LIN {X -0.033,Y -190.233,Z 1843.877,A 0.000,B 0.000,C 90.000,E1 337.922} C_DIS
LIN {X -0.106,Y -193.186,Z 1843.850,A 0.000,B 0.000,C 90.000,E1 332.999} C_DIS
LIN {X 0.019,Y -196.283,Z 1843.827,A 0.000,B 0.000,C 90.000,E1 328.869} C_DIS
LIN {X -0.019,Y -199.902,Z 1843.804,A 0.000,B 0.000,C 90.000,E1 324.815} C_DIS
LIN {X -0.088,Y -204.049,Z 1843.782,A 0.000,B 0.000,C 90.000,E1 320.803} C_DIS
LIN {X 0.012,Y -209.249,Z 1843.760,A 0.000,B 0.000,C 90.000,E1 316.782} C_DIS
LIN {X -0.006,Y -211.916,Z 1843.751,A 0.000,B 0.000,C 90.000,E1 315.202} C_DIS
LIN {X 0.008,Y -215.116,Z 1843.742,A 0.000,B 0.000,C 90.000,E1 313.623} C_DIS
LIN {X -0.083,Y -218.974,Z 1843.734,A 0.000,B 0.000,C 90.000,E1 312.081} C_DIS
LIN {X -0.117,Y -223.654,Z 1843.725,A 0.000,B 0.000,C 90.000,E1 310.539} C_DIS
LIN {X -0.067,Y -229.271,Z 1843.717,A 0.000,B 0.000,C 90.000,E1 308.991} C_DIS
LIN {X 0.059,Y -235.659,Z 1843.708,A 0.000,B 0.000,C 90.000,E1 307.443} C_DIS
LIN {X -0.053,Y -246.348,Z 1843.696,A 0.000,B 0.000,C 90.000,E1 305.231} C_DIS
LIN {X -0.015,Y -260.231,Z 1843.682,A 0.000,B 0.000,C 90.000,E1 302.673} C_DIS
LIN {X -0.147,Y -278.257,Z 1843.666,A 0.000,B 0.000,C 90.000,E1 299.873} C_DIS
LIN {X -0.079,Y -294.898,Z 1843.652,A 0.000,B 0.000,C 90.000,E1 297.462} C_DIS
LIN {X -0.078,Y -306.901,Z 1843.643,A 0.000,B 0.000,C 90.000,E1 295.796} C_DIS
LIN {X -0.041,Y -323.612,Z 1843.631,A 0.000,B 0.000,C 90.000,E1 293.515} C_DIS
LIN {X 0.188,Y -333.099,Z 1843.624,A 0.000,B 0.000,C 90.000,E1 292.206} C_DIS
LIN {X 0.104,Y -342.269,Z 1843.617,A 0.000,B 0.000,C 90.000,E1 290.972} C_DIS
LIN {X 0.010,Y -350.803,Z 1843.610,A 0.000,B 0.000,C 90.000,E1 289.758} C_DIS
LIN {X -0.017,Y -356.794,Z 1843.605,A 0.000,B 0.000,C 90.000,E1 288.852} C_DIS
LIN {X 0.008,Y -362.167,Z 1843.600,A 0.000,B 0.000,C 90.000,E1 287.946} C_DIS
LIN {X 0.020,Y -365.351,Z 1843.596,A 0.000,B 0.000,C 90.000,E1 287.347} C_DIS
LIN {X 0.131,Y -369.387,Z 1843.591,A 0.000,B 0.000,C 90.000,E1 286.441} C_DIS
LIN {X 0.190,Y -371.679,Z 1843.588,A 0.000,B 0.000,C 90.000,E1 285.843} C_DIS
LIN {X -0.108,Y -374.517,Z 1843.583,A 0.000,B 0.000,C 90.000,E1 285.009} C_DIS
LIN {X -0.025,Y -375.965,Z 1843.580,A 0.000,B 0.000,C 90.000,E1 284.411} C_DIS
LIN {X -0.024,Y -376.991,Z 1843.577,A 0.000,B 0.000,C 90.000,E1 283.828} C_DIS
LIN {X -0.010,Y -377.620,Z 1843.574,A 0.000,B 0.000,C 90.000,E1 283.244} C_DIS
LIN {X 0.094,Y -377.791,Z 1843.570,A 0.000,B 0.000,C 90.000,E1 282.647} C_DIS
LIN {X 0.119,Y -377.552,Z 1843.567,A 0.000,B 0.000,C 90.000,E1 282.063} C_DIS
LIN {X 0.145,Y -376.875,Z 1843.564,A 0.000,B 0.000,C 90.000,E1 281.478} C_DIS
LIN {X 0.170,Y -375.718,Z 1843.561,A 0.000,B 0.000,C 90.000,E1 280.894} C_DIS
LIN {X 0.190,Y -374.108,Z 1843.557,A 0.000,B 0.000,C 90.000,E1 280.310} C_DIS
LIN {X 0.139,Y -370.889,Z 1843.553,A 0.000,B 0.000,C 90.000,E1 279.443} C_DIS
LIN {X -0.018,Y -362.561,Z 1843.541,A 0.000,B 0.000,C 90.000,E1 277.409} C_DIS
LIN {X 0.184,Y -358.290,Z 1843.536,A 0.000,B 0.000,C 90.000,E1 276.486} C_DIS
LIN {X 0.048,Y -354.814,Z 1843.533,A 0.000,B 0.000,C 90.000,E1 275.910} C_DIS
LIN {X -0.105,Y -350.748,Z 1843.530,A 0.000,B 0.000,C 90.000,E1 275.334} C_DIS
LIN {X 0.069,Y -345.924,Z 1843.526,A 0.000,B 0.000,C 90.000,E1 274.702} C_DIS
LIN {X -0.112,Y -340.429,Z 1843.523,A 0.000,B 0.000,C 90.000,E1 274.131} C_DIS
LIN {X -0.087,Y -334.526,Z 1843.520,A 0.000,B 0.000,C 90.000,E1 273.555} C_DIS
LIN {X -0.114,Y -328.400,Z 1843.517,A 0.000,B 0.000,C 90.000,E1 273.037} C_DIS
LIN {X 0.077,Y -322.038,Z 1843.514,A 0.000,B 0.000,C 90.000,E1 272.522} C_DIS
LIN {X -0.131,Y -315.451,Z 1843.512,A 0.000,B 0.000,C 90.000,E1 272.121} C_DIS
LIN {X -0.025,Y -308.681,Z 1843.510,A 0.000,B 0.000,C 90.000,E1 271.718} C_DIS
LIN {X 0.079,Y -301.563,Z 1843.508,A 0.000,B 0.000,C 90.000,E1 271.375} C_DIS
LIN {X -0.137,Y -294.097,Z 1843.506,A 0.000,B 0.000,C 90.000,E1 271.146} C_DIS
LIN {X -0.063,Y -286.185,Z 1843.505,A 0.000,B 0.000,C 90.000,E1 270.917} C_DIS
LIN {X 0.097,Y -271.303,Z 1843.503,A 0.000,B 0.000,C 90.000,E1 270.573} C_DIS
LIN {X 0.056,Y -249.540,Z 1843.501,A 0.000,B 0.000,C 90.000,E1 270.172} C_DIS
LIN {X -0.017,Y -240.784,Z 1843.500,A 0.000,B 0.000,C 90.000,E1 270.057} C_DIS
LIN {X 0.111,Y -230.998,Z 1843.500,A 0.000,B 0.000,C 90.000,E1 269.943} C_DIS
LIN {X 0.068,Y -181.555,Z 1843.500,A 0.000,B 0.000,C 90.000,E1 269.943} C_DIS
LIN {X -0.012,Y -180.816,Z 1843.471,A 0.000,B 0.000,C 90.000,E1 264.837} C_DIS
LIN {X 0.065,Y -178.919,Z 1843.443,A 0.000,B 0.000,C 90.000,E1 259.746} C_DIS
LIN {X -0.026,Y -175.964,Z 1843.415,A 0.000,B 0.000,C 90.000,E1 254.685} C_DIS
LIN {X 0.090,Y -175.441,Z 1843.410,A 0.000,B 0.000,C 90.000,E1 253.795} C_DIS
LIN {X -0.069,Y -172.198,Z 1843.386,A 0.000,B 0.000,C 90.000,E1 249.571} C_DIS
LIN {X -0.092,Y -171.671,Z 1843.382,A 0.000,B 0.000,C 90.000,E1 248.720} C_DIS
LIN {X -0.100,Y -167.896,Z 1843.358,A 0.000,B 0.000,C 90.000,E1 244.409} C_DIS
LIN {X 0.068,Y -166.636,Z 1843.348,A 0.000,B 0.000,C 90.000,E1 242.615} C_DIS
LIN {X -0.026,Y -162.621,Z 1843.324,A 0.000,B 0.000,C 90.000,E1 238.280} C_DIS
LIN {X 0.033,Y -161.307,Z 1843.314,A 0.000,B 0.000,C 90.000,E1 236.501} C_DIS
LIN {X -0.057,Y -157.304,Z 1843.289,A 0.000,B 0.000,C 90.000,E1 232.110} C_DIS
LIN {X 0.096,Y -155.281,Z 1843.275,A 0.000,B 0.000,C 90.000,E1 229.380} C_DIS
LIN {X 0.024,Y -151.646,Z 1843.250,A 0.000,B 0.000,C 90.000,E1 224.919} C_DIS
LIN {X -0.040,Y -150.514,Z 1843.240,A 0.000,B 0.000,C 90.000,E1 223.137} C_DIS
LIN {X -0.016,Y -147.239,Z 1843.214,A 0.000,B 0.000,C 90.000,E1 218.588} C_DIS
LIN {X -0.050,Y -145.263,Z 1843.194,A 0.000,B 0.000,C 90.000,E1 214.945} C_DIS
LIN {X -0.016,Y -142.373,Z 1843.163,A 0.000,B 0.000,C 90.000,E1 209.411} C_DIS
LIN {X -0.021,Y -141.757,Z 1843.153,A 0.000,B 0.000,C 90.000,E1 207.564} C_DIS
LIN {X 0.030,Y -139.498,Z 1843.117,A 0.000,B 0.000,C 90.000,E1 201.046} C_DIS
LIN {X 0.067,Y -139.004,Z 1843.101,A 0.000,B 0.000,C 90.000,E1 198.236} C_DIS
LIN {X 0.023,Y -138.339,Z 1843.055,A 0.000,B 0.000,C 90.000,E1 189.849} C_DIS
LIN {X 0.046,Y -139.406,Z 1843.008,A 0.000,B 0.000,C 90.000,E1 181.432} C_DIS
LIN {X -0.041,Y -141.314,Z 1842.972,A 0.000,B 0.000,C 90.000,E1 174.951} C_DIS
LIN {X 0.057,Y -142.673,Z 1842.956,A 0.000,B 0.000,C 90.000,E1 172.129} C_DIS
LIN {X 0.038,Y -145.026,Z 1842.931,A 0.000,B 0.000,C 90.000,E1 167.521} C_DIS
LIN {X -0.005,Y -147.652,Z 1842.910,A 0.000,B 0.000,C 90.000,E1 163.866} C_DIS
LIN {X -0.070,Y -150.288,Z 1842.890,A 0.000,B 0.000,C 90.000,E1 160.242} C_DIS
LIN {X -0.057,Y -153.695,Z 1842.870,A 0.000,B 0.000,C 90.000,E1 156.613} C_DIS
LIN {X -0.003,Y -157.109,Z 1842.850,A 0.000,B 0.000,C 90.000,E1 152.999} C_DIS
LIN {X 0.074,Y -161.250,Z 1842.830,A 0.000,B 0.000,C 90.000,E1 149.410} C_DIS
LIN {X 0.020,Y -163.337,Z 1842.820,A 0.000,B 0.000,C 90.000,E1 147.661} C_DIS
LIN {X 0.027,Y -167.791,Z 1842.801,A 0.000,B 0.000,C 90.000,E1 144.149} C_DIS
LIN {X 0.043,Y -171.605,Z 1842.786,A 0.000,B 0.000,C 90.000,E1 141.537} C_DIS
LIN {X 0.091,Y -176.559,Z 1842.767,A 0.000,B 0.000,C 90.000,E1 138.081} C_DIS
LIN {X -0.036,Y -180.857,Z 1842.753,A 0.000,B 0.000,C 90.000,E1 135.567} C_DIS
LIN {X -0.052,Y -186.270,Z 1842.734,A 0.000,B 0.000,C 90.000,E1 132.204} C_DIS
LIN {X 0.007,Y -190.905,Z 1842.720,A 0.000,B 0.000,C 90.000,E1 129.688} C_DIS
LIN {X 0.076,Y -196.671,Z 1842.702,A 0.000,B 0.000,C 90.000,E1 126.377} C_DIS
LIN {X -0.006,Y -199.914,Z 1842.693,A 0.000,B 0.000,C 90.000,E1 124.771} C_DIS
LIN {X 0.024,Y -204.306,Z 1842.680,A 0.000,B 0.000,C 90.000,E1 122.339} C_DIS
LIN {X -0.011,Y -210.652,Z 1842.662,A 0.000,B 0.000,C 90.000,E1 119.155} C_DIS
LIN {X 0.093,Y -216.474,Z 1842.644,A 0.000,B 0.000,C 90.000,E1 115.976} C_DIS
LIN {X -0.090,Y -219.587,Z 1842.636,A 0.000,B 0.000,C 90.000,E1 114.463} C_DIS
LIN {X -0.088,Y -224.053,Z 1842.622,A 0.000,B 0.000,C 90.000,E1 111.897} C_DIS
LIN {X 0.120,Y -283.246,Z 1842.621,A 0.000,B 0.000,C 90.000,E1 111.844} C_DIS
LIN {X 0.108,Y -287.787,Z 1842.621,A 0.000,B 0.000,C 90.000,E1 111.716} C_DIS
LIN {X 0.096,Y -289.851,Z 1842.620,A 0.000,B 0.000,C 90.000,E1 111.589} C_DIS
LIN {X -0.038,Y -292.673,Z 1842.619,A 0.000,B 0.000,C 90.000,E1 111.354} C_DIS
LIN {X 0.109,Y -296.409,Z 1842.616,A 0.000,B 0.000,C 90.000,E1 110.791} C_DIS
LIN {X 0.006,Y -309.662,Z 1842.603,A 0.000,B 0.000,C 90.000,E1 108.489} C_DIS
LIN {X 0.117,Y -324.275,Z 1842.590,A 0.000,B 0.000,C 90.000,E1 106.205} C_DIS
LIN {X -0.145,Y -337.983,Z 1842.580,A 0.000,B 0.000,C 90.000,E1 104.356} C_DIS
LIN {X 0.012,Y -352.877,Z 1842.569,A 0.000,B 0.000,C 90.000,E1 102.479} C_DIS
LIN {X 0.073,Y -371.270,Z 1842.558,A 0.000,B 0.000,C 90.000,E1 100.433} C_DIS
LIN {X 0.155,Y -390.141,Z 1842.548,A 0.000,B 0.000,C 90.000,E1 98.568} C_DIS
LIN {X 0.107,Y -409.354,Z 1842.538,A 0.000,B 0.000,C 90.000,E1 96.891} C_DIS
LIN {X -0.048,Y -431.732,Z 1842.529,A 0.000,B 0.000,C 90.000,E1 95.163} C_DIS
LIN {X 0.106,Y -440.040,Z 1842.525,A 0.000,B 0.000,C 90.000,E1 94.531} C_DIS
LIN {X -0.059,Y -443.726,Z 1842.523,A 0.000,B 0.000,C 90.000,E1 94.131} C_DIS
LIN {X 0.140,Y -445.289,Z 1842.521,A 0.000,B 0.000,C 90.000,E1 93.841} C_DIS
LIN {X -0.135,Y -446.467,Z 1842.520,A 0.000,B 0.000,C 90.000,E1 93.612} C_DIS
LIN {X -0.184,Y -447.912,Z 1842.517,A 0.000,B 0.000,C 90.000,E1 93.094} C_DIS
LIN {X 0.197,Y -448.360,Z 1842.514,A 0.000,B 0.000,C 90.000,E1 92.522} C_DIS
LIN {X 0.143,Y -447.881,Z 1842.511,A 0.000,B 0.000,C 90.000,E1 92.007} C_DIS
LIN {X 0.105,Y -446.408,Z 1842.508,A 0.000,B 0.000,C 90.000,E1 91.489} C_DIS
LIN {X -0.145,Y -445.226,Z 1842.507,A 0.000,B 0.000,C 90.000,E1 91.260} C_DIS
LIN {X 0.067,Y -435.424,Z 1842.498,A 0.000,B 0.000,C 90.000,E1 89.656} C_DIS
LIN {X 0.113,Y -425.490,Z 1842.489,A 0.000,B 0.000,C 90.000,E1 88.051} C_DIS
LIN {X 0.084,Y -413.715,Z 1842.479,A 0.000,B 0.000,C 90.000,E1 86.159} C_DIS
LIN {X -0.136,Y -401.847,Z 1842.468,A 0.000,B 0.000,C 90.000,E1 84.261} C_DIS
LIN {X -0.146,Y -389.902,Z 1842.457,A 0.000,B 0.000,C 90.000,E1 82.299} C_DIS
LIN {X 0.018,Y -377.966,Z 1842.446,A 0.000,B 0.000,C 90.000,E1 80.274} C_DIS
LIN {X -0.003,Y -361.271,Z 1842.430,A 0.000,B 0.000,C 90.000,E1 77.353} C_DIS
LIN {X 0.075,Y -345.625,Z 1842.413,A 0.000,B 0.000,C 90.000,E1 74.338} C_DIS
LIN {X 0.111,Y -333.627,Z 1842.399,A 0.000,B 0.000,C 90.000,E1 71.873} C_DIS
LIN {X -0.034,Y -321.887,Z 1842.385,A 0.000,B 0.000,C 90.000,E1 69.390} C_DIS
LIN {X 0.090,Y -309.231,Z 1842.370,A 0.000,B 0.000,C 90.000,E1 66.485} C_DIS
LIN {X 0.059,Y -299.647,Z 1842.357,A 0.000,B 0.000,C 90.000,E1 64.204} C_DIS
LIN {X -0.060,Y -287.547,Z 1842.340,A 0.000,B 0.000,C 90.000,E1 61.229} C_DIS
LIN {X -0.147,Y -278.152,Z 1842.327,A 0.000,B 0.000,C 90.000,E1 58.869} C_DIS
LIN {X -0.011,Y -268.705,Z 1842.313,A 0.000,B 0.000,C 90.000,E1 56.421} C_DIS
LIN {X -0.059,Y -260.529,Z 1842.302,A 0.000,B 0.000,C 90.000,E1 54.322} C_DIS
LIN {X -0.106,Y -252.310,Z 1842.290,A 0.000,B 0.000,C 90.000,E1 52.190} C_DIS
LIN {X -0.005,Y -242.722,Z 1842.276,A 0.000,B 0.000,C 90.000,E1 49.622} C_DIS
LIN {X 0.011,Y -233.304,Z 1842.261,A 0.000,B 0.000,C 90.000,E1 47.025} C_DIS
LIN {X -0.098,Y -222.999,Z 1842.245,A 0.000,B 0.000,C 90.000,E1 44.028} C_DIS
LIN {X 0.023,Y -213.186,Z 1842.227,A 0.000,B 0.000,C 90.000,E1 40.906} C_DIS
LIN {X 0.101,Y -204.177,Z 1842.210,A 0.000,B 0.000,C 90.000,E1 37.729} C_DIS
LIN {X -0.043,Y -200.670,Z 1842.202,A 0.000,B 0.000,C 90.000,E1 36.423} C_DIS
LIN {X 0.097,Y -200.694,Z 1842.202,A 0.000,B 0.000,C 90.000,E1 36.377} C_DIS
LIN {X -0.009,Y -207.756,Z 1842.196,A 0.000,B 0.000,C 90.000,E1 35.358} C_DIS
LIN {X 0.040,Y -209.524,Z 1842.194,A 0.000,B 0.000,C 90.000,E1 34.945} C_DIS
LIN {X 0.089,Y -210.171,Z 1842.192,A 0.000,B 0.000,C 90.000,E1 34.532} C_DIS
LIN {X -0.072,Y -210.542,Z 1842.188,A 0.000,B 0.000,C 90.000,E1 33.785} C_DIS
LIN {X 0.063,Y -210.374,Z 1842.183,A 0.000,B 0.000,C 90.000,E1 32.959} C_DIS
LIN {X 0.041,Y -209.330,Z 1842.174,A 0.000,B 0.000,C 90.000,E1 31.386} C_DIS
LIN {X 0.077,Y -207.876,Z 1842.166,A 0.000,B 0.000,C 90.000,E1 29.795} C_DIS
LIN {X -0.004,Y -205.334,Z 1842.152,A 0.000,B 0.000,C 90.000,E1 27.436} C_DIS
LIN {X -0.011,Y -200.959,Z 1842.130,A 0.000,B 0.000,C 90.000,E1 23.439} C_DIS
LIN {X 0.017,Y -197.151,Z 1842.108,A 0.000,B 0.000,C 90.000,E1 19.396} C_DIS
LIN {X -0.078,Y -193.232,Z 1842.081,A 0.000,B 0.000,C 90.000,E1 14.537} C_DIS
LIN {X 0.049,Y -189.554,Z 1842.049,A 0.000,B 0.000,C 90.000,E1 8.746} C_DIS
LIN {X -0.048,Y -187.048,Z 1842.016,A 0.000,B 0.000,C 90.000,E1 2.980} C_DIS
LIN {X -0.043,Y -185.845,Z 1841.988,A 0.000,B 0.000,C 90.000,E1 357.879} C_DIS
LIN {X 0.070,Y -185.626,Z 1841.956,A 0.000,B 0.000,C 90.000,E1 352.008} C_DIS
LIN {X 0.075,Y -186.651,Z 1841.923,A 0.000,B 0.000,C 90.000,E1 346.172} C_DIS
LIN {X -0.055,Y -188.055,Z 1841.900,A 0.000,B 0.000,C 90.000,E1 342.054} C_DIS
LIN {X 0.061,Y -190.369,Z 1841.873,A 0.000,B 0.000,C 90.000,E1 337.050} C_DIS
LIN {X 0.079,Y -193.498,Z 1841.845,A 0.000,B 0.000,C 90.000,E1 332.103} C_DIS
LIN {X -0.026,Y -196.711,Z 1841.822,A 0.000,B 0.000,C 90.000,E1 328.043} C_DIS
LIN {X -0.050,Y -200.488,Z 1841.800,A 0.000,B 0.000,C 90.000,E1 323.989} C_DIS
LIN {X -0.009,Y -204.833,Z 1841.777,A 0.000,B 0.000,C 90.000,E1 319.952} C_DIS
LIN {X 0.051,Y -209.167,Z 1841.760,A 0.000,B 0.000,C 90.000,E1 316.743} C_DIS
LIN {X 0.116,Y -213.426,Z 1841.747,A 0.000,B 0.000,C 90.000,E1 314.352} C_DIS
LIN {X -0.100,Y -217.998,Z 1841.736,A 0.000,B 0.000,C 90.000,E1 312.447} C_DIS
LIN {X 0.018,Y -222.547,Z 1841.727,A 0.000,B 0.000,C 90.000,E1 310.862} C_DIS
LIN {X -0.054,Y -226.536,Z 1841.721,A 0.000,B 0.000,C 90.000,E1 309.725} C_DIS
LIN {X 0.036,Y -232.619,Z 1841.712,A 0.000,B 0.000,C 90.000,E1 308.177} C_DIS
LIN {X 0.037,Y -241.159,Z 1841.702,A 0.000,B 0.000,C 90.000,E1 306.297} C_DIS
LIN {X -0.115,Y -252.461,Z 1841.689,A 0.000,B 0.000,C 90.000,E1 304.119} C_DIS
LIN {X -0.022,Y -262.758,Z 1841.679,A 0.000,B 0.000,C 90.000,E1 302.291} C_DIS
LIN {X 0.059,Y -281.021,Z 1841.664,A 0.000,B 0.000,C 90.000,E1 299.461} C_DIS
LIN {X 0.069,Y -297.771,Z 1841.651,A 0.000,B 0.000,C 90.000,E1 297.078} C_DIS
LIN {X 0.115,Y -309.796,Z 1841.641,A 0.000,B 0.000,C 90.000,E1 295.412} C_DIS
LIN {X -0.137,Y -324.198,Z 1841.630,A 0.000,B 0.000,C 90.000,E1 293.515} C_DIS
LIN {X 0.097,Y -333.737,Z 1841.623,A 0.000,B 0.000,C 90.000,E1 292.206} C_DIS
LIN {X 0.018,Y -342.918,Z 1841.617,A 0.000,B 0.000,C 90.000,E1 290.972} C_DIS
LIN {X -0.070,Y -351.484,Z 1841.610,A 0.000,B 0.000,C 90.000,E1 289.758} C_DIS
LIN {X -0.092,Y -357.481,Z 1841.605,A 0.000,B 0.000,C 90.000,E1 288.852} C_DIS
LIN {X -0.061,Y -362.841,Z 1841.600,A 0.000,B 0.000,C 90.000,E1 287.946} C_DIS
LIN {X 0.064,Y -366.038,Z 1841.596,A 0.000,B 0.000,C 90.000,E1 287.330} C_DIS
LIN {X 0.098,Y -368.830,Z 1841.593,A 0.000,B 0.000,C 90.000,E1 286.732} C_DIS
LIN {X 0.134,Y -372.332,Z 1841.588,A 0.000,B 0.000,C 90.000,E1 285.843} C_DIS
LIN {X -0.160,Y -375.103,Z 1841.583,A 0.000,B 0.000,C 90.000,E1 285.009} C_DIS
LIN {X -0.072,Y -376.527,Z 1841.580,A 0.000,B 0.000,C 90.000,E1 284.411} C_DIS
LIN {X -0.068,Y -377.488,Z 1841.577,A 0.000,B 0.000,C 90.000,E1 283.828} C_DIS
LIN {X -0.051,Y -378.135,Z 1841.573,A 0.000,B 0.000,C 90.000,E1 283.244} C_DIS
LIN {X 0.057,Y -378.299,Z 1841.570,A 0.000,B 0.000,C 90.000,E1 282.647} C_DIS
LIN {X 0.085,Y -377.992,Z 1841.567,A 0.000,B 0.000,C 90.000,E1 282.063} C_DIS
LIN {X 0.114,Y -377.277,Z 1841.564,A 0.000,B 0.000,C 90.000,E1 281.478} C_DIS
LIN {X 0.141,Y -376.078,Z 1841.561,A 0.000,B 0.000,C 90.000,E1 280.894} C_DIS
LIN {X 0.164,Y -374.447,Z 1841.557,A 0.000,B 0.000,C 90.000,E1 280.310} C_DIS
LIN {X 0.177,Y -372.370,Z 1841.554,A 0.000,B 0.000,C 90.000,E1 279.726} C_DIS
LIN {X -0.034,Y -362.799,Z 1841.541,A 0.000,B 0.000,C 90.000,E1 277.409} C_DIS
LIN {X 0.171,Y -358.476,Z 1841.536,A 0.000,B 0.000,C 90.000,E1 276.486} C_DIS
LIN {X 0.035,Y -355.006,Z 1841.533,A 0.000,B 0.000,C 90.000,E1 275.910} C_DIS
LIN {X -0.115,Y -350.943,Z 1841.530,A 0.000,B 0.000,C 90.000,E1 275.334} C_DIS
LIN {X 0.059,Y -346.104,Z 1841.526,A 0.000,B 0.000,C 90.000,E1 274.702} C_DIS
LIN {X -0.110,Y -340.587,Z 1841.523,A 0.000,B 0.000,C 90.000,E1 274.131} C_DIS
LIN {X -0.072,Y -334.680,Z 1841.520,A 0.000,B 0.000,C 90.000,E1 273.555} C_DIS
LIN {X -0.044,Y -328.746,Z 1841.517,A 0.000,B 0.000,C 90.000,E1 273.037} C_DIS
LIN {X -0.104,Y -322.559,Z 1841.514,A 0.000,B 0.000,C 90.000,E1 272.579} C_DIS
LIN {X 0.028,Y -316.078,Z 1841.512,A 0.000,B 0.000,C 90.000,E1 272.121} C_DIS
LIN {X 0.142,Y -309.263,Z 1841.510,A 0.000,B 0.000,C 90.000,E1 271.718} C_DIS
LIN {X -0.094,Y -302.144,Z 1841.508,A 0.000,B 0.000,C 90.000,E1 271.432} C_DIS
LIN {X -0.058,Y -294.567,Z 1841.506,A 0.000,B 0.000,C 90.000,E1 271.146} C_DIS
LIN {X 0.003,Y -286.661,Z 1841.505,A 0.000,B 0.000,C 90.000,E1 270.917} C_DIS
LIN {X -0.131,Y -271.712,Z 1841.503,A 0.000,B 0.000,C 90.000,E1 270.630} C_DIS
LIN {X 0.114,Y -250.110,Z 1841.501,A 0.000,B 0.000,C 90.000,E1 270.172} C_DIS
LIN {X 0.028,Y -241.287,Z 1841.500,A 0.000,B 0.000,C 90.000,E1 270.057} C_DIS
LIN {X -0.085,Y -231.549,Z 1841.500,A 0.000,B 0.000,C 90.000,E1 270.000} C_DIS
LIN {X -0.087,Y -181.556,Z 1841.500,A 0.000,B 0.000,C 90.000,E1 270.000} C_DIS
LIN {X 0.013,Y -180.819,Z 1841.471,A 0.000,B 0.000,C 90.000,E1 264.837} C_DIS
LIN {X 0.088,Y -178.922,Z 1841.443,A 0.000,B 0.000,C 90.000,E1 259.746} C_DIS
LIN {X -0.002,Y -175.968,Z 1841.415,A 0.000,B 0.000,C 90.000,E1 254.685} C_DIS
LIN {X -0.054,Y -175.448,Z 1841.410,A 0.000,B 0.000,C 90.000,E1 253.850} C_DIS
LIN {X -0.045,Y -172.202,Z 1841.386,A 0.000,B 0.000,C 90.000,E1 249.571} C_DIS
LIN {X -0.068,Y -171.677,Z 1841.382,A 0.000,B 0.000,C 90.000,E1 248.720} C_DIS
LIN {X -0.077,Y -167.903,Z 1841.358,A 0.000,B 0.000,C 90.000,E1 244.409} C_DIS
LIN {X -0.058,Y -166.642,Z 1841.348,A 0.000,B 0.000,C 90.000,E1 242.666} C_DIS
LIN {X -0.003,Y -162.628,Z 1841.324,A 0.000,B 0.000,C 90.000,E1 238.280} C_DIS
LIN {X 0.056,Y -161.315,Z 1841.314,A 0.000,B 0.000,C 90.000,E1 236.501} C_DIS
LIN {X -0.034,Y -157.311,Z 1841.289,A 0.000,B 0.000,C 90.000,E1 232.110} C_DIS
LIN {X -0.101,Y -155.289,Z 1841.275,A 0.000,B 0.000,C 90.000,E1 229.461} C_DIS
LIN {X 0.046,Y -151.651,Z 1841.250,A 0.000,B 0.000,C 90.000,E1 224.919} C_DIS
LIN {X -0.018,Y -150.519,Z 1841.240,A 0.000,B 0.000,C 90.000,E1 223.137} C_DIS
LIN {X 0.006,Y -147.243,Z 1841.214,A 0.000,B 0.000,C 90.000,E1 218.588} C_DIS
LIN {X -0.029,Y -145.268,Z 1841.194,A 0.000,B 0.000,C 90.000,E1 214.945} C_DIS
LIN {X 0.005,Y -142.377,Z 1841.163,A 0.000,B 0.000,C 90.000,E1 209.411} C_DIS
LIN {X 0.054,Y -141.352,Z 1841.148,A 0.000,B 0.000,C 90.000,E1 206.616} C_DIS
LIN {X 0.038,Y -139.339,Z 1841.112,A 0.000,B 0.000,C 90.000,E1 200.120} C_DIS
LIN {X -0.044,Y -139.007,Z 1841.102,A 0.000,B 0.000,C 90.000,E1 198.290} C_DIS
LIN {X 0.044,Y -138.339,Z 1841.055,A 0.000,B 0.000,C 90.000,E1 189.849} C_DIS
LIN {X 0.066,Y -139.403,Z 1841.008,A 0.000,B 0.000,C 90.000,E1 181.432} C_DIS
LIN {X -0.020,Y -141.310,Z 1840.972,A 0.000,B 0.000,C 90.000,E1 174.951} C_DIS
LIN {X -0.063,Y -142.670,Z 1840.956,A 0.000,B 0.000,C 90.000,E1 172.186} C_DIS
LIN {X 0.059,Y -145.020,Z 1840.931,A 0.000,B 0.000,C 90.000,E1 167.521} C_DIS
LIN {X 0.017,Y -147.647,Z 1840.910,A 0.000,B 0.000,C 90.000,E1 163.866} C_DIS
LIN {X -0.048,Y -150.281,Z 1840.890,A 0.000,B 0.000,C 90.000,E1 160.242} C_DIS
LIN {X -0.036,Y -153.686,Z 1840.870,A 0.000,B 0.000,C 90.000,E1 156.613} C_DIS
LIN {X 0.020,Y -157.101,Z 1840.850,A 0.000,B 0.000,C 90.000,E1 152.999} C_DIS
LIN {X -0.042,Y -161.240,Z 1840.830,A 0.000,B 0.000,C 90.000,E1 149.459} C_DIS
LIN {X 0.044,Y -163.327,Z 1840.820,A 0.000,B 0.000,C 90.000,E1 147.661} C_DIS
LIN {X -0.086,Y -167.780,Z 1840.801,A 0.000,B 0.000,C 90.000,E1 144.196} C_DIS
LIN {X 0.065,Y -171.595,Z 1840.786,A 0.000,B 0.000,C 90.000,E1 141.537} C_DIS
LIN {X -0.003,Y -176.547,Z 1840.767,A 0.000,B 0.000,C 90.000,E1 138.119} C_DIS
LIN {X -0.011,Y -180.846,Z 1840.753,A 0.000,B 0.000,C 90.000,E1 135.567} C_DIS
LIN {X -0.027,Y -186.256,Z 1840.734,A 0.000,B 0.000,C 90.000,E1 132.204} C_DIS
LIN {X -0.089,Y -190.893,Z 1840.721,A 0.000,B 0.000,C 90.000,E1 129.725} C_DIS
LIN {X -0.057,Y -196.657,Z 1840.702,A 0.000,B 0.000,C 90.000,E1 126.423} C_DIS
LIN {X 0.019,Y -199.899,Z 1840.693,A 0.000,B 0.000,C 90.000,E1 124.771} C_DIS
LIN {X 0.050,Y -204.292,Z 1840.680,A 0.000,B 0.000,C 90.000,E1 122.339} C_DIS
LIN {X 0.017,Y -210.640,Z 1840.662,A 0.000,B 0.000,C 90.000,E1 119.155} C_DIS
LIN {X 0.120,Y -216.459,Z 1840.645,A 0.000,B 0.000,C 90.000,E1 115.976} C_DIS
LIN {X -0.063,Y -219.576,Z 1840.636,A 0.000,B 0.000,C 90.000,E1 114.463} C_DIS
LIN {X -0.086,Y -224.052,Z 1840.622,A 0.000,B 0.000,C 90.000,E1 111.897} C_DIS
LIN {X 0.119,Y -283.485,Z 1840.621,A 0.000,B 0.000,C 90.000,E1 111.844} C_DIS
LIN {X 0.043,Y -286.450,Z 1840.621,A 0.000,B 0.000,C 90.000,E1 111.791} C_DIS
LIN {X -0.061,Y -290.264,Z 1840.620,A 0.000,B 0.000,C 90.000,E1 111.589} C_DIS
LIN {X -0.002,Y -292.614,Z 1840.619,A 0.000,B 0.000,C 90.000,E1 111.354} C_DIS
LIN {X 0.089,Y -296.429,Z 1840.616,A 0.000,B 0.000,C 90.000,E1 110.791} C_DIS
LIN {X -0.015,Y -309.684,Z 1840.603,A 0.000,B 0.000,C 90.000,E1 108.489} C_DIS
LIN {X 0.095,Y -324.299,Z 1840.590,A 0.000,B 0.000,C 90.000,E1 106.205} C_DIS
LIN {X 0.160,Y -338.009,Z 1840.580,A 0.000,B 0.000,C 90.000,E1 104.300} C_DIS
LIN {X -0.011,Y -352.906,Z 1840.569,A 0.000,B 0.000,C 90.000,E1 102.479} C_DIS
LIN {X 0.052,Y -371.300,Z 1840.558,A 0.000,B 0.000,C 90.000,E1 100.433} C_DIS
LIN {X 0.135,Y -390.172,Z 1840.548,A 0.000,B 0.000,C 90.000,E1 98.568} C_DIS
LIN {X 0.087,Y -409.385,Z 1840.538,A 0.000,B 0.000,C 90.000,E1 96.891} C_DIS
LIN {X -0.067,Y -431.764,Z 1840.529,A 0.000,B 0.000,C 90.000,E1 95.163} C_DIS
LIN {X 0.089,Y -440.063,Z 1840.525,A 0.000,B 0.000,C 90.000,E1 94.531} C_DIS
LIN {X -0.085,Y -443.740,Z 1840.523,A 0.000,B 0.000,C 90.000,E1 94.131} C_DIS
LIN {X 0.114,Y -445.298,Z 1840.521,A 0.000,B 0.000,C 90.000,E1 93.841} C_DIS
LIN {X -0.161,Y -446.470,Z 1840.520,A 0.000,B 0.000,C 90.000,E1 93.612} C_DIS
LIN {X -0.211,Y -447.907,Z 1840.517,A 0.000,B 0.000,C 90.000,E1 93.094} C_DIS
LIN {X 0.170,Y -448.346,Z 1840.514,A 0.000,B 0.000,C 90.000,E1 92.522} C_DIS
LIN {X 0.117,Y -447.860,Z 1840.511,A 0.000,B 0.000,C 90.000,E1 92.007} C_DIS
LIN {X 0.079,Y -446.378,Z 1840.508,A 0.000,B 0.000,C 90.000,E1 91.489} C_DIS
LIN {X -0.171,Y -445.190,Z 1840.507,A 0.000,B 0.000,C 90.000,E1 91.260} C_DIS
LIN {X 0.040,Y -435.384,Z 1840.498,A 0.000,B 0.000,C 90.000,E1 89.656} C_DIS
LIN {X 0.086,Y -425.450,Z 1840.489,A 0.000,B 0.000,C 90.000,E1 88.051} C_DIS
LIN {X 0.057,Y -413.674,Z 1840.479,A 0.000,B 0.000,C 90.000,E1 86.159} C_DIS
LIN {X -0.163,Y -401.804,Z 1840.468,A 0.000,B 0.000,C 90.000,E1 84.261} C_DIS
LIN {X -0.173,Y -389.860,Z 1840.457,A 0.000,B 0.000,C 90.000,E1 82.299} C_DIS
LIN {X -0.009,Y -377.924,Z 1840.446,A 0.000,B 0.000,C 90.000,E1 80.274} C_DIS
LIN {X -0.030,Y -361.229,Z 1840.430,A 0.000,B 0.000,C 90.000,E1 77.353} C_DIS
LIN {X 0.048,Y -345.584,Z 1840.413,A 0.000,B 0.000,C 90.000,E1 74.338} C_DIS
LIN {X 0.084,Y -333.587,Z 1840.399,A 0.000,B 0.000,C 90.000,E1 71.873} C_DIS
LIN {X -0.061,Y -321.843,Z 1840.385,A 0.000,B 0.000,C 90.000,E1 69.390} C_DIS
LIN {X 0.063,Y -309.189,Z 1840.369,A 0.000,B 0.000,C 90.000,E1 66.485} C_DIS
LIN {X 0.032,Y -299.603,Z 1840.357,A 0.000,B 0.000,C 90.000,E1 64.204} C_DIS
LIN {X 0.165,Y -287.502,Z 1840.340,A 0.000,B 0.000,C 90.000,E1 61.179} C_DIS
LIN {X 0.063,Y -278.109,Z 1840.327,A 0.000,B 0.000,C 90.000,E1 58.820} C_DIS
LIN {X -0.037,Y -268.663,Z 1840.313,A 0.000,B 0.000,C 90.000,E1 56.421} C_DIS
LIN {X -0.086,Y -260.488,Z 1840.302,A 0.000,B 0.000,C 90.000,E1 54.322} C_DIS
LIN {X -0.134,Y -252.268,Z 1840.290,A 0.000,B 0.000,C 90.000,E1 52.190} C_DIS
LIN {X -0.032,Y -242.682,Z 1840.276,A 0.000,B 0.000,C 90.000,E1 49.622} C_DIS
LIN {X -0.015,Y -233.263,Z 1840.261,A 0.000,B 0.000,C 90.000,E1 47.025} C_DIS
LIN {X -0.124,Y -222.959,Z 1840.244,A 0.000,B 0.000,C 90.000,E1 44.028} C_DIS
LIN {X -0.003,Y -213.149,Z 1840.227,A 0.000,B 0.000,C 90.000,E1 40.906} C_DIS
LIN {X 0.041,Y -207.133,Z 1840.216,A 0.000,B 0.000,C 90.000,E1 38.830} C_DIS
LIN {X 0.018,Y -207.134,Z 1840.216,A 0.000,B 0.000,C 90.000,E1 38.830} C_DIS
LIN {X 0.080,Y -213.958,Z 1840.210,A 0.000,B 0.000,C 90.000,E1 37.729} C_DIS
LIN {X -0.022,Y -215.625,Z 1840.208,A 0.000,B 0.000,C 90.000,E1 37.363} C_DIS
LIN {X 0.049,Y -216.231,Z 1840.205,A 0.000,B 0.000,C 90.000,E1 36.950} C_DIS
LIN {X 0.044,Y -216.542,Z 1840.201,A 0.000,B 0.000,C 90.000,E1 36.171} C_DIS
LIN {X 0.044,Y -216.336,Z 1840.197,A 0.000,B 0.000,C 90.000,E1 35.391} C_DIS
LIN {X 0.045,Y -215.875,Z 1840.192,A 0.000,B 0.000,C 90.000,E1 34.612} C_DIS
LIN {X -0.083,Y -214.421,Z 1840.184,A 0.000,B 0.000,C 90.000,E1 33.086} C_DIS
LIN {X -0.009,Y -211.580,Z 1840.171,A 0.000,B 0.000,C 90.000,E1 30.718} C_DIS
LIN {X -0.019,Y -208.525,Z 1840.157,A 0.000,B 0.000,C 90.000,E1 28.359} C_DIS
LIN {X 0.087,Y -204.417,Z 1840.140,A 0.000,B 0.000,C 90.000,E1 25.155} C_DIS
LIN {X -0.002,Y -199.841,Z 1840.118,A 0.000,B 0.000,C 90.000,E1 21.173} C_DIS
LIN {X -0.007,Y -195.216,Z 1840.091,A 0.000,B 0.000,C 90.000,E1 16.315} C_DIS
LIN {X -0.055,Y -191.961,Z 1840.068,A 0.000,B 0.000,C 90.000,E1 12.243} C_DIS
LIN {X -0.035,Y -188.799,Z 1840.041,A 0.000,B 0.000,C 90.000,E1 7.296} C_DIS
LIN {X 0.000,Y -185.857,Z 1840.000,A 0.000,B 0.000,C 90.000,E1 360.000} C_DIS
LIN {X -0.057,Y -185.209,Z 1839.960,A 0.000,B 0.000,C 90.000,E1 352.875} C_DIS
LIN {X -0.100,Y -185.876,Z 1839.932,A 0.000,B 0.000,C 90.000,E1 347.881} C_DIS
LIN {X 0.010,Y -187.386,Z 1839.905,A 0.000,B 0.000,C 90.000,E1 342.851} C_DIS
LIN {X 0.096,Y -189.614,Z 1839.877,A 0.000,B 0.000,C 90.000,E1 337.847} C_DIS
LIN {X 0.012,Y -192.673,Z 1839.850,A 0.000,B 0.000,C 90.000,E1 332.922} C_DIS
LIN {X 0.057,Y -196.472,Z 1839.822,A 0.000,B 0.000,C 90.000,E1 327.995} C_DIS
LIN {X 0.137,Y -200.267,Z 1839.800,A 0.000,B 0.000,C 90.000,E1 323.909} C_DIS
LIN {X 0.046,Y -204.669,Z 1839.777,A 0.000,B 0.000,C 90.000,E1 319.908} C_DIS
LIN {X -0.107,Y -207.861,Z 1839.764,A 0.000,B 0.000,C 90.000,E1 317.553} C_DIS
LIN {X -0.073,Y -211.874,Z 1839.751,A 0.000,B 0.000,C 90.000,E1 315.162} C_DIS
LIN {X 0.092,Y -215.166,Z 1839.742,A 0.000,B 0.000,C 90.000,E1 313.542} C_DIS
LIN {X 0.002,Y -219.151,Z 1839.733,A 0.000,B 0.000,C 90.000,E1 312.000} C_DIS
LIN {X -0.029,Y -223.984,Z 1839.725,A 0.000,B 0.000,C 90.000,E1 310.458} C_DIS
LIN {X 0.088,Y -228.205,Z 1839.718,A 0.000,B 0.000,C 90.000,E1 309.277} C_DIS
LIN {X 0.017,Y -236.158,Z 1839.708,A 0.000,B 0.000,C 90.000,E1 307.397} C_DIS
LIN {X -0.081,Y -246.969,Z 1839.695,A 0.000,B 0.000,C 90.000,E1 305.185} C_DIS
LIN {X -0.023,Y -261.007,Z 1839.681,A 0.000,B 0.000,C 90.000,E1 302.625} C_DIS
LIN {X 0.011,Y -279.137,Z 1839.666,A 0.000,B 0.000,C 90.000,E1 299.795} C_DIS
LIN {X 0.104,Y -295.862,Z 1839.652,A 0.000,B 0.000,C 90.000,E1 297.385} C_DIS
LIN {X 0.011,Y -310.339,Z 1839.641,A 0.000,B 0.000,C 90.000,E1 295.412} C_DIS
LIN {X 0.112,Y -324.721,Z 1839.630,A 0.000,B 0.000,C 90.000,E1 293.462} C_DIS
LIN {X 0.054,Y -334.287,Z 1839.623,A 0.000,B 0.000,C 90.000,E1 292.206} C_DIS
LIN {X -0.018,Y -343.514,Z 1839.616,A 0.000,B 0.000,C 90.000,E1 290.972} C_DIS
LIN {X -0.101,Y -352.126,Z 1839.610,A 0.000,B 0.000,C 90.000,E1 289.758} C_DIS
LIN {X -0.117,Y -358.117,Z 1839.605,A 0.000,B 0.000,C 90.000,E1 288.852} C_DIS
LIN {X -0.080,Y -363.491,Z 1839.600,A 0.000,B 0.000,C 90.000,E1 287.946} C_DIS
LIN {X 0.048,Y -366.680,Z 1839.596,A 0.000,B 0.000,C 90.000,E1 287.330} C_DIS
LIN {X 0.086,Y -369.481,Z 1839.593,A 0.000,B 0.000,C 90.000,E1 286.732} C_DIS
LIN {X 0.128,Y -372.939,Z 1839.588,A 0.000,B 0.000,C 90.000,E1 285.843} C_DIS
LIN {X -0.160,Y -375.680,Z 1839.583,A 0.000,B 0.000,C 90.000,E1 285.009} C_DIS
LIN {X -0.069,Y -377.065,Z 1839.580,A 0.000,B 0.000,C 90.000,E1 284.411} C_DIS
LIN {X -0.061,Y -378.030,Z 1839.577,A 0.000,B 0.000,C 90.000,E1 283.828} C_DIS
LIN {X -0.041,Y -378.647,Z 1839.573,A 0.000,B 0.000,C 90.000,E1 283.244} C_DIS
LIN {X 0.071,Y -378.770,Z 1839.570,A 0.000,B 0.000,C 90.000,E1 282.647} C_DIS
LIN {X 0.101,Y -378.462,Z 1839.567,A 0.000,B 0.000,C 90.000,E1 282.063} C_DIS
LIN {X 0.133,Y -377.701,Z 1839.564,A 0.000,B 0.000,C 90.000,E1 281.478} C_DIS
LIN {X 0.164,Y -376.483,Z 1839.561,A 0.000,B 0.000,C 90.000,E1 280.894} C_DIS
LIN {X 0.189,Y -374.806,Z 1839.557,A 0.000,B 0.000,C 90.000,E1 280.310} C_DIS
LIN {X 0.204,Y -372.713,Z 1839.554,A 0.000,B 0.000,C 90.000,E1 279.726} C_DIS
LIN {X 0.025,Y -364.353,Z 1839.543,A 0.000,B 0.000,C 90.000,E1 277.701} C_DIS
LIN {X -0.109,Y -360.307,Z 1839.538,A 0.000,B 0.000,C 90.000,E1 276.834} C_DIS
LIN {X 0.124,Y -357.051,Z 1839.535,A 0.000,B 0.000,C 90.000,E1 276.201} C_DIS
LIN {X -0.015,Y -353.268,Z 1839.531,A 0.000,B 0.000,C 90.000,E1 275.625} C_DIS
LIN {X -0.171,Y -348.796,Z 1839.528,A 0.000,B 0.000,C 90.000,E1 275.049} C_DIS
LIN {X -0.007,Y -343.634,Z 1839.525,A 0.000,B 0.000,C 90.000,E1 274.416} C_DIS
LIN {X -0.135,Y -337.769,Z 1839.521,A 0.000,B 0.000,C 90.000,E1 273.841} C_DIS
LIN {X -0.071,Y -328.831,Z 1839.517,A 0.000,B 0.000,C 90.000,E1 273.037} C_DIS
LIN {X 0.159,Y -322.525,Z 1839.514,A 0.000,B 0.000,C 90.000,E1 272.522} C_DIS
LIN {X -0.027,Y -315.992,Z 1839.512,A 0.000,B 0.000,C 90.000,E1 272.121} C_DIS
LIN {X 0.089,Y -309.189,Z 1839.510,A 0.000,B 0.000,C 90.000,E1 271.718} C_DIS
LIN {X -0.138,Y -302.062,Z 1839.508,A 0.000,B 0.000,C 90.000,E1 271.432} C_DIS
LIN {X -0.069,Y -294.406,Z 1839.506,A 0.000,B 0.000,C 90.000,E1 271.146} C_DIS
LIN {X 0.013,Y -286.689,Z 1839.505,A 0.000,B 0.000,C 90.000,E1 270.917} C_DIS
LIN {X -0.064,Y -275.367,Z 1839.504,A 0.000,B 0.000,C 90.000,E1 270.688} C_DIS
LIN {X -0.118,Y -250.134,Z 1839.501,A 0.000,B 0.000,C 90.000,E1 270.229} C_DIS
LIN {X 0.049,Y -241.308,Z 1839.500,A 0.000,B 0.000,C 90.000,E1 270.057} C_DIS
LIN {X -0.037,Y -232.641,Z 1839.500,A 0.000,B 0.000,C 90.000,E1 270.000} C_DIS
LIN {X -0.063,Y -229.892,Z 1839.500,A 0.000,B 0.000,C 90.000,E1 270.000} C_DIS
LIN {X -0.070,Y -181.557,Z 1839.500,A 0.000,B 0.000,C 90.000,E1 270.000} C_DIS
LIN {X 0.033,Y -180.821,Z 1839.471,A 0.000,B 0.000,C 90.000,E1 264.837} C_DIS
LIN {X -0.067,Y -178.924,Z 1839.443,A 0.000,B 0.000,C 90.000,E1 259.803} C_DIS
LIN {X -0.028,Y -175.971,Z 1839.415,A 0.000,B 0.000,C 90.000,E1 254.700} C_DIS
LIN {X -0.034,Y -175.454,Z 1839.410,A 0.000,B 0.000,C 90.000,E1 253.850} C_DIS
LIN {X -0.026,Y -172.206,Z 1839.386,A 0.000,B 0.000,C 90.000,E1 249.571} C_DIS
LIN {X -0.047,Y -171.681,Z 1839.382,A 0.000,B 0.000,C 90.000,E1 248.720} C_DIS
LIN {X -0.057,Y -167.908,Z 1839.358,A 0.000,B 0.000,C 90.000,E1 244.409} C_DIS
LIN {X -0.038,Y -166.649,Z 1839.348,A 0.000,B 0.000,C 90.000,E1 242.666} C_DIS
LIN {X 0.016,Y -162.632,Z 1839.324,A 0.000,B 0.000,C 90.000,E1 238.280} C_DIS
LIN {X 0.076,Y -161.320,Z 1839.314,A 0.000,B 0.000,C 90.000,E1 236.501} C_DIS
LIN {X -0.016,Y -157.316,Z 1839.289,A 0.000,B 0.000,C 90.000,E1 232.110} C_DIS
LIN {X -0.083,Y -155.296,Z 1839.275,A 0.000,B 0.000,C 90.000,E1 229.461} C_DIS
LIN {X 0.065,Y -151.656,Z 1839.250,A 0.000,B 0.000,C 90.000,E1 224.919} C_DIS
LIN {X 0.001,Y -150.524,Z 1839.240,A 0.000,B 0.000,C 90.000,E1 223.137} C_DIS
LIN {X 0.024,Y -147.248,Z 1839.214,A 0.000,B 0.000,C 90.000,E1 218.588} C_DIS
LIN {X -0.011,Y -145.273,Z 1839.194,A 0.000,B 0.000,C 90.000,E1 214.945} C_DIS
LIN {X 0.023,Y -142.379,Z 1839.163,A 0.000,B 0.000,C 90.000,E1 209.411} C_DIS
LIN {X 0.073,Y -141.355,Z 1839.148,A 0.000,B 0.000,C 90.000,E1 206.616} C_DIS
LIN {X 0.056,Y -139.341,Z 1839.112,A 0.000,B 0.000,C 90.000,E1 200.120} C_DIS
LIN {X -0.026,Y -139.009,Z 1839.102,A 0.000,B 0.000,C 90.000,E1 198.290} C_DIS
LIN {X 0.061,Y -138.340,Z 1839.055,A 0.000,B 0.000,C 90.000,E1 189.849} C_DIS
LIN {X -0.055,Y -139.402,Z 1839.008,A 0.000,B 0.000,C 90.000,E1 181.489} C_DIS
LIN {X -0.002,Y -141.306,Z 1838.972,A 0.000,B 0.000,C 90.000,E1 174.951} C_DIS
LIN {X -0.044,Y -142.668,Z 1838.957,A 0.000,B 0.000,C 90.000,E1 172.186} C_DIS
LIN {X 0.077,Y -145.016,Z 1838.931,A 0.000,B 0.000,C 90.000,E1 167.521} C_DIS
LIN {X 0.035,Y -147.642,Z 1838.910,A 0.000,B 0.000,C 90.000,E1 163.866} C_DIS
LIN {X -0.030,Y -150.276,Z 1838.890,A 0.000,B 0.000,C 90.000,E1 160.242} C_DIS
LIN {X -0.016,Y -153.679,Z 1838.870,A 0.000,B 0.000,C 90.000,E1 156.613} C_DIS
LIN {X 0.040,Y -157.093,Z 1838.850,A 0.000,B 0.000,C 90.000,E1 152.999} C_DIS
LIN {X -0.023,Y -161.231,Z 1838.830,A 0.000,B 0.000,C 90.000,E1 149.459} C_DIS
LIN {X 0.063,Y -163.319,Z 1838.820,A 0.000,B 0.000,C 90.000,E1 147.661} C_DIS
LIN {X -0.066,Y -167.771,Z 1838.801,A 0.000,B 0.000,C 90.000,E1 144.196} C_DIS
LIN {X 0.086,Y -171.586,Z 1838.786,A 0.000,B 0.000,C 90.000,E1 141.537} C_DIS
LIN {X 0.017,Y -176.536,Z 1838.767,A 0.000,B 0.000,C 90.000,E1 138.119} C_DIS
LIN {X 0.010,Y -180.835,Z 1838.753,A 0.000,B 0.000,C 90.000,E1 135.567} C_DIS
LIN {X -0.006,Y -186.244,Z 1838.734,A 0.000,B 0.000,C 90.000,E1 132.204} C_DIS
LIN {X -0.068,Y -190.881,Z 1838.721,A 0.000,B 0.000,C 90.000,E1 129.725} C_DIS
LIN {X -0.036,Y -196.645,Z 1838.702,A 0.000,B 0.000,C 90.000,E1 126.423} C_DIS
LIN {X 0.042,Y -199.885,Z 1838.693,A 0.000,B 0.000,C 90.000,E1 124.771} C_DIS
LIN {X 0.073,Y -204.280,Z 1838.680,A 0.000,B 0.000,C 90.000,E1 122.339} C_DIS
LIN {X 0.039,Y -210.630,Z 1838.662,A 0.000,B 0.000,C 90.000,E1 119.155} C_DIS
LIN {X -0.051,Y -216.448,Z 1838.645,A 0.000,B 0.000,C 90.000,E1 116.027} C_DIS
LIN {X -0.040,Y -219.566,Z 1838.636,A 0.000,B 0.000,C 90.000,E1 114.463} C_DIS
LIN {X -0.090,Y -224.055,Z 1838.622,A 0.000,B 0.000,C 90.000,E1 111.897} C_DIS
LIN {X 0.114,Y -283.757,Z 1838.621,A 0.000,B 0.000,C 90.000,E1 111.844} C_DIS
LIN {X 0.072,Y -286.325,Z 1838.621,A 0.000,B 0.000,C 90.000,E1 111.791} C_DIS
LIN {X -0.031,Y -290.198,Z 1838.620,A 0.000,B 0.000,C 90.000,E1 111.589} C_DIS
LIN {X 0.028,Y -292.564,Z 1838.619,A 0.000,B 0.000,C 90.000,E1 111.354} C_DIS
LIN {X 0.135,Y -296.378,Z 1838.616,A 0.000,B 0.000,C 90.000,E1 110.791} C_DIS
LIN {X 0.032,Y -309.630,Z 1838.603,A 0.000,B 0.000,C 90.000,E1 108.489} C_DIS
LIN {X -0.169,Y -324.239,Z 1838.590,A 0.000,B 0.000,C 90.000,E1 106.260} C_DIS
LIN {X -0.118,Y -337.944,Z 1838.580,A 0.000,B 0.000,C 90.000,E1 104.356} C_DIS
LIN {X 0.039,Y -352.836,Z 1838.569,A 0.000,B 0.000,C 90.000,E1 102.479} C_DIS
LIN {X 0.099,Y -371.228,Z 1838.558,A 0.000,B 0.000,C 90.000,E1 100.433} C_DIS
LIN {X 0.180,Y -390.098,Z 1838.548,A 0.000,B 0.000,C 90.000,E1 98.568} C_DIS
LIN {X 0.131,Y -409.310,Z 1838.538,A 0.000,B 0.000,C 90.000,E1 96.891} C_DIS
LIN {X -0.026,Y -431.688,Z 1838.529,A 0.000,B 0.000,C 90.000,E1 95.163} C_DIS
LIN {X 0.129,Y -439.999,Z 1838.525,A 0.000,B 0.000,C 90.000,E1 94.531} C_DIS
LIN {X -0.035,Y -443.688,Z 1838.523,A 0.000,B 0.000,C 90.000,E1 94.131} C_DIS
LIN {X 0.165,Y -445.254,Z 1838.521,A 0.000,B 0.000,C 90.000,E1 93.841} C_DIS
LIN {X -0.111,Y -446.434,Z 1838.520,A 0.000,B 0.000,C 90.000,E1 93.612} C_DIS
LIN {X -0.160,Y -447.882,Z 1838.517,A 0.000,B 0.000,C 90.000,E1 93.094} C_DIS
LIN {X 0.222,Y -448.333,Z 1838.514,A 0.000,B 0.000,C 90.000,E1 92.522} C_DIS
LIN {X 0.167,Y -447.856,Z 1838.511,A 0.000,B 0.000,C 90.000,E1 92.007} C_DIS
LIN {X 0.129,Y -446.387,Z 1838.508,A 0.000,B 0.000,C 90.000,E1 91.489} C_DIS
LIN {X -0.120,Y -445.207,Z 1838.507,A 0.000,B 0.000,C 90.000,E1 91.260} C_DIS
LIN {X 0.089,Y -435.404,Z 1838.498,A 0.000,B 0.000,C 90.000,E1 89.656} C_DIS
LIN {X 0.135,Y -425.474,Z 1838.489,A 0.000,B 0.000,C 90.000,E1 88.051} C_DIS
LIN {X 0.105,Y -413.697,Z 1838.479,A 0.000,B 0.000,C 90.000,E1 86.159} C_DIS
LIN {X -0.115,Y -401.827,Z 1838.468,A 0.000,B 0.000,C 90.000,E1 84.261} C_DIS
LIN {X -0.127,Y -389.883,Z 1838.457,A 0.000,B 0.000,C 90.000,E1 82.299} C_DIS
LIN {X 0.036,Y -377.947,Z 1838.446,A 0.000,B 0.000,C 90.000,E1 80.274} C_DIS
LIN {X 0.014,Y -361.247,Z 1838.430,A 0.000,B 0.000,C 90.000,E1 77.353} C_DIS
LIN {X 0.090,Y -345.600,Z 1838.413,A 0.000,B 0.000,C 90.000,E1 74.338} C_DIS
LIN {X 0.125,Y -333.600,Z 1838.399,A 0.000,B 0.000,C 90.000,E1 71.873} C_DIS
LIN {X -0.021,Y -321.856,Z 1838.385,A 0.000,B 0.000,C 90.000,E1 69.390} C_DIS
LIN {X 0.102,Y -309.200,Z 1838.370,A 0.000,B 0.000,C 90.000,E1 66.485} C_DIS
LIN {X 0.070,Y -299.610,Z 1838.357,A 0.000,B 0.000,C 90.000,E1 64.204} C_DIS
LIN {X -0.050,Y -287.508,Z 1838.340,A 0.000,B 0.000,C 90.000,E1 61.229} C_DIS
LIN {X -0.139,Y -278.116,Z 1838.327,A 0.000,B 0.000,C 90.000,E1 58.869} C_DIS
LIN {X -0.004,Y -268.671,Z 1838.313,A 0.000,B 0.000,C 90.000,E1 56.421} C_DIS
LIN {X -0.052,Y -260.498,Z 1838.302,A 0.000,B 0.000,C 90.000,E1 54.322} C_DIS
LIN {X -0.101,Y -252.279,Z 1838.290,A 0.000,B 0.000,C 90.000,E1 52.190} C_DIS
LIN {X -0.001,Y -242.692,Z 1838.276,A 0.000,B 0.000,C 90.000,E1 49.622} C_DIS
LIN {X 0.015,Y -233.272,Z 1838.261,A 0.000,B 0.000,C 90.000,E1 47.025} C_DIS
LIN {X -0.095,Y -222.966,Z 1838.245,A 0.000,B 0.000,C 90.000,E1 44.028} C_DIS
LIN {X 0.006,Y -213.872,Z 1838.229,A 0.000,B 0.000,C 90.000,E1 41.148} C_DIS
LIN {X -0.017,Y -213.868,Z 1838.229,A 0.000,B 0.000,C 90.000,E1 41.148} C_DIS
LIN {X -0.024,Y -219.873,Z 1838.223,A 0.000,B 0.000,C 90.000,E1 40.135} C_DIS
LIN {X 0.061,Y -221.779,Z 1838.221,A 0.000,B 0.000,C 90.000,E1 39.725} C_DIS
LIN {X -0.024,Y -222.481,Z 1838.219,A 0.000,B 0.000,C 90.000,E1 39.358} C_DIS
LIN {X -0.027,Y -222.812,Z 1838.214,A 0.000,B 0.000,C 90.000,E1 38.588} C_DIS
LIN {X 0.008,Y -222.549,Z 1838.210,A 0.000,B 0.000,C 90.000,E1 37.810} C_DIS
LIN {X -0.089,Y -221.231,Z 1838.202,A 0.000,B 0.000,C 90.000,E1 36.297} C_DIS
LIN {X -0.124,Y -218.467,Z 1838.189,A 0.000,B 0.000,C 90.000,E1 33.992} C_DIS
LIN {X 0.033,Y -215.119,Z 1838.176,A 0.000,B 0.000,C 90.000,E1 31.623} C_DIS
LIN {X 0.054,Y -210.453,Z 1838.158,A 0.000,B 0.000,C 90.000,E1 28.487} C_DIS
LIN {X 0.108,Y -204.809,Z 1838.136,A 0.000,B 0.000,C 90.000,E1 24.515} C_DIS
LIN {X -0.052,Y -199.954,Z 1838.114,A 0.000,B 0.000,C 90.000,E1 20.556} C_DIS
LIN {X 0.067,Y -195.057,Z 1838.087,A 0.000,B 0.000,C 90.000,E1 15.662} C_DIS
LIN {X -0.032,Y -190.969,Z 1838.060,A 0.000,B 0.000,C 90.000,E1 10.782} C_DIS
LIN {X -0.007,Y -187.279,Z 1838.028,A 0.000,B 0.000,C 90.000,E1 4.992} C_DIS
LIN {X 0.025,Y -184.924,Z 1837.984,A 0.000,B 0.000,C 90.000,E1 357.020} C_DIS
LIN {X -0.054,Y -184.963,Z 1837.951,A 0.000,B 0.000,C 90.000,E1 351.197} C_DIS
LIN {X -0.001,Y -186.194,Z 1837.919,A 0.000,B 0.000,C 90.000,E1 345.338} C_DIS
LIN {X -0.077,Y -188.047,Z 1837.891,A 0.000,B 0.000,C 90.000,E1 340.369} C_DIS
LIN {X 0.066,Y -190.731,Z 1837.863,A 0.000,B 0.000,C 90.000,E1 335.357} C_DIS
LIN {X 0.011,Y -193.573,Z 1837.840,A 0.000,B 0.000,C 90.000,E1 331.257} C_DIS
LIN {X 0.008,Y -196.944,Z 1837.818,A 0.000,B 0.000,C 90.000,E1 327.168} C_DIS
LIN {X -0.061,Y -200.904,Z 1837.795,A 0.000,B 0.000,C 90.000,E1 323.130} C_DIS
LIN {X -0.012,Y -205.525,Z 1837.773,A 0.000,B 0.000,C 90.000,E1 319.094} C_DIS
LIN {X -0.013,Y -209.019,Z 1837.759,A 0.000,B 0.000,C 90.000,E1 316.701} C_DIS
LIN {X 0.115,Y -211.867,Z 1837.751,A 0.000,B 0.000,C 90.000,E1 315.081} C_DIS
LIN {X -0.022,Y -215.205,Z 1837.742,A 0.000,B 0.000,C 90.000,E1 313.542} C_DIS
LIN {X -0.114,Y -219.287,Z 1837.733,A 0.000,B 0.000,C 90.000,E1 312.000} C_DIS
LIN {X -0.069,Y -222.865,Z 1837.727,A 0.000,B 0.000,C 90.000,E1 310.825} C_DIS
LIN {X 0.033,Y -226.942,Z 1837.720,A 0.000,B 0.000,C 90.000,E1 309.644} C_DIS
LIN {X 0.086,Y -234.730,Z 1837.710,A 0.000,B 0.000,C 90.000,E1 307.729} C_DIS
LIN {X -0.042,Y -245.393,Z 1837.697,A 0.000,B 0.000,C 90.000,E1 305.518} C_DIS
LIN {X 0.097,Y -257.236,Z 1837.685,A 0.000,B 0.000,C 90.000,E1 303.293} C_DIS
LIN {X -0.090,Y -268.007,Z 1837.675,A 0.000,B 0.000,C 90.000,E1 301.544} C_DIS
LIN {X 0.032,Y -284.269,Z 1837.662,A 0.000,B 0.000,C 90.000,E1 299.077} C_DIS
LIN {X -0.013,Y -298.761,Z 1837.650,A 0.000,B 0.000,C 90.000,E1 297.052} C_DIS
LIN {X -0.060,Y -313.305,Z 1837.639,A 0.000,B 0.000,C 90.000,E1 295.079} C_DIS
LIN {X 0.038,Y -327.811,Z 1837.629,A 0.000,B 0.000,C 90.000,E1 293.131} C_DIS
LIN {X -0.141,Y -339.702,Z 1837.620,A 0.000,B 0.000,C 90.000,E1 291.589} C_DIS
LIN {X 0.174,Y -348.626,Z 1837.613,A 0.000,B 0.000,C 90.000,E1 290.301} C_DIS
LIN {X 0.128,Y -354.947,Z 1837.608,A 0.000,B 0.000,C 90.000,E1 289.396} C_DIS
LIN {X 0.137,Y -360.705,Z 1837.603,A 0.000,B 0.000,C 90.000,E1 288.489} C_DIS
LIN {X -0.096,Y -364.212,Z 1837.599,A 0.000,B 0.000,C 90.000,E1 287.928} C_DIS
LIN {X -0.076,Y -367.385,Z 1837.596,A 0.000,B 0.000,C 90.000,E1 287.330} C_DIS
LIN {X -0.035,Y -370.172,Z 1837.593,A 0.000,B 0.000,C 90.000,E1 286.732} C_DIS
LIN {X 0.013,Y -373.602,Z 1837.588,A 0.000,B 0.000,C 90.000,E1 285.843} C_DIS
LIN {X 0.094,Y -376.306,Z 1837.583,A 0.000,B 0.000,C 90.000,E1 284.954} C_DIS
LIN {X 0.190,Y -377.649,Z 1837.580,A 0.000,B 0.000,C 90.000,E1 284.356} C_DIS
LIN {X -0.163,Y -378.568,Z 1837.577,A 0.000,B 0.000,C 90.000,E1 283.828} C_DIS
LIN {X -0.141,Y -379.134,Z 1837.573,A 0.000,B 0.000,C 90.000,E1 283.244} C_DIS
LIN {X -0.025,Y -379.236,Z 1837.570,A 0.000,B 0.000,C 90.000,E1 282.647} C_DIS
LIN {X 0.009,Y -378.902,Z 1837.567,A 0.000,B 0.000,C 90.000,E1 282.063} C_DIS
LIN {X 0.044,Y -378.114,Z 1837.564,A 0.000,B 0.000,C 90.000,E1 281.478} C_DIS
LIN {X 0.077,Y -376.868,Z 1837.561,A 0.000,B 0.000,C 90.000,E1 280.894} C_DIS
LIN {X 0.104,Y -375.147,Z 1837.557,A 0.000,B 0.000,C 90.000,E1 280.310} C_DIS
LIN {X 0.065,Y -371.808,Z 1837.552,A 0.000,B 0.000,C 90.000,E1 279.443} C_DIS
LIN {X -0.048,Y -364.596,Z 1837.543,A 0.000,B 0.000,C 90.000,E1 277.701} C_DIS
LIN {X 0.179,Y -360.503,Z 1837.538,A 0.000,B 0.000,C 90.000,E1 276.777} C_DIS
LIN {X 0.057,Y -357.165,Z 1837.535,A 0.000,B 0.000,C 90.000,E1 276.201} C_DIS
LIN {X -0.080,Y -353.393,Z 1837.531,A 0.000,B 0.000,C 90.000,E1 275.625} C_DIS
LIN {X 0.111,Y -348.893,Z 1837.528,A 0.000,B 0.000,C 90.000,E1 274.992} C_DIS
LIN {X -0.069,Y -343.665,Z 1837.524,A 0.000,B 0.000,C 90.000,E1 274.416} C_DIS
LIN {X 0.151,Y -337.850,Z 1837.521,A 0.000,B 0.000,C 90.000,E1 273.784} C_DIS
LIN {X -0.029,Y -331.811,Z 1837.518,A 0.000,B 0.000,C 90.000,E1 273.269} C_DIS
LIN {X 0.067,Y -325.597,Z 1837.515,A 0.000,B 0.000,C 90.000,E1 272.751} C_DIS
LIN {X 0.073,Y -319.043,Z 1837.513,A 0.000,B 0.000,C 90.000,E1 272.293} C_DIS
LIN {X 0.056,Y -312.397,Z 1837.511,A 0.000,B 0.000,C 90.000,E1 271.892} C_DIS
LIN {X 0.010,Y -305.351,Z 1837.509,A 0.000,B 0.000,C 90.000,E1 271.547} C_DIS
LIN {X 0.010,Y -298.388,Z 1837.507,A 0.000,B 0.000,C 90.000,E1 271.260} C_DIS
LIN {X -0.062,Y -290.518,Z 1837.506,A 0.000,B 0.000,C 90.000,E1 271.031} C_DIS
LIN {X 0.025,Y -279.146,Z 1837.504,A 0.000,B 0.000,C 90.000,E1 270.745} C_DIS
LIN {X -0.089,Y -253.606,Z 1837.501,A 0.000,B 0.000,C 90.000,E1 270.286} C_DIS
LIN {X 0.036,Y -240.960,Z 1837.500,A 0.000,B 0.000,C 90.000,E1 270.057} C_DIS
LIN {X 0.007,Y -233.460,Z 1837.500,A 0.000,B 0.000,C 90.000,E1 270.000} C_DIS
LIN {X -0.039,Y -228.868,Z 1837.500,A 0.000,B 0.000,C 90.000,E1 270.000} C_DIS
LIN {X -0.049,Y -181.558,Z 1837.500,A 0.000,B 0.000,C 90.000,E1 270.000} C_DIS
LIN {X 0.060,Y -180.823,Z 1837.471,A 0.000,B 0.000,C 90.000,E1 264.837} C_DIS
LIN {X -0.039,Y -178.927,Z 1837.443,A 0.000,B 0.000,C 90.000,E1 259.803} C_DIS
LIN {X -0.001,Y -175.975,Z 1837.415,A 0.000,B 0.000,C 90.000,E1 254.700} C_DIS
LIN {X -0.056,Y -175.461,Z 1837.410,A 0.000,B 0.000,C 90.000,E1 253.866} C_DIS
LIN {X 0.001,Y -172.212,Z 1837.386,A 0.000,B 0.000,C 90.000,E1 249.571} C_DIS
LIN {X -0.021,Y -171.688,Z 1837.382,A 0.000,B 0.000,C 90.000,E1 248.720} C_DIS
LIN {X -0.030,Y -167.915,Z 1837.358,A 0.000,B 0.000,C 90.000,E1 244.409} C_DIS
LIN {X -0.011,Y -166.656,Z 1837.348,A 0.000,B 0.000,C 90.000,E1 242.666} C_DIS
LIN {X 0.042,Y -162.640,Z 1837.324,A 0.000,B 0.000,C 90.000,E1 238.280} C_DIS
LIN {X -0.033,Y -161.328,Z 1837.314,A 0.000,B 0.000,C 90.000,E1 236.548} C_DIS
LIN {X 0.010,Y -157.323,Z 1837.290,A 0.000,B 0.000,C 90.000,E1 232.110} C_DIS
LIN {X -0.057,Y -155.304,Z 1837.275,A 0.000,B 0.000,C 90.000,E1 229.461} C_DIS
LIN {X -0.018,Y -151.662,Z 1837.250,A 0.000,B 0.000,C 90.000,E1 224.960} C_DIS
LIN {X 0.026,Y -150.529,Z 1837.240,A 0.000,B 0.000,C 90.000,E1 223.137} C_DIS
LIN {X -0.044,Y -147.254,Z 1837.214,A 0.000,B 0.000,C 90.000,E1 218.624} C_DIS
LIN {X 0.014,Y -145.280,Z 1837.194,A 0.000,B 0.000,C 90.000,E1 214.945} C_DIS
LIN {X 0.046,Y -142.383,Z 1837.163,A 0.000,B 0.000,C 90.000,E1 209.411} C_DIS
LIN {X -0.031,Y -141.360,Z 1837.148,A 0.000,B 0.000,C 90.000,E1 206.668} C_DIS
LIN {X -0.052,Y -139.343,Z 1837.112,A 0.000,B 0.000,C 90.000,E1 200.174} C_DIS
LIN {X -0.047,Y -139.012,Z 1837.102,A 0.000,B 0.000,C 90.000,E1 198.308} C_DIS
LIN {X -0.052,Y -138.341,Z 1837.055,A 0.000,B 0.000,C 90.000,E1 189.905} C_DIS
LIN {X -0.032,Y -139.399,Z 1837.008,A 0.000,B 0.000,C 90.000,E1 181.489} C_DIS
LIN {X 0.022,Y -141.302,Z 1836.972,A 0.000,B 0.000,C 90.000,E1 174.951} C_DIS
LIN {X -0.021,Y -142.664,Z 1836.957,A 0.000,B 0.000,C 90.000,E1 172.186} C_DIS
LIN {X -0.071,Y -145.010,Z 1836.931,A 0.000,B 0.000,C 90.000,E1 167.589} C_DIS
LIN {X 0.060,Y -147.636,Z 1836.911,A 0.000,B 0.000,C 90.000,E1 163.866} C_DIS
LIN {X -0.005,Y -150.268,Z 1836.890,A 0.000,B 0.000,C 90.000,E1 160.242} C_DIS
LIN {X 0.009,Y -153.669,Z 1836.870,A 0.000,B 0.000,C 90.000,E1 156.613} C_DIS
LIN {X 0.065,Y -157.083,Z 1836.850,A 0.000,B 0.000,C 90.000,E1 152.999} C_DIS
LIN {X 0.004,Y -161.219,Z 1836.830,A 0.000,B 0.000,C 90.000,E1 149.459} C_DIS
LIN {X -0.049,Y -163.309,Z 1836.821,A 0.000,B 0.000,C 90.000,E1 147.709} C_DIS
LIN {X -0.040,Y -167.758,Z 1836.801,A 0.000,B 0.000,C 90.000,E1 144.196} C_DIS
LIN {X -0.022,Y -171.574,Z 1836.786,A 0.000,B 0.000,C 90.000,E1 141.582} C_DIS
LIN {X -0.087,Y -176.522,Z 1836.767,A 0.000,B 0.000,C 90.000,E1 138.162} C_DIS
LIN {X 0.038,Y -180.820,Z 1836.753,A 0.000,B 0.000,C 90.000,E1 135.567} C_DIS
LIN {X 0.022,Y -186.229,Z 1836.734,A 0.000,B 0.000,C 90.000,E1 132.204} C_DIS
LIN {X -0.039,Y -190.867,Z 1836.721,A 0.000,B 0.000,C 90.000,E1 129.725} C_DIS
LIN {X -0.006,Y -196.628,Z 1836.702,A 0.000,B 0.000,C 90.000,E1 126.423} C_DIS
LIN {X -0.093,Y -199.868,Z 1836.693,A 0.000,B 0.000,C 90.000,E1 124.818} C_DIS
LIN {X 0.102,Y -204.264,Z 1836.680,A 0.000,B 0.000,C 90.000,E1 122.339} C_DIS
LIN {X 0.069,Y -210.615,Z 1836.662,A 0.000,B 0.000,C 90.000,E1 119.155} C_DIS
LIN {X -0.021,Y -216.431,Z 1836.645,A 0.000,B 0.000,C 90.000,E1 116.027} C_DIS
LIN {X -0.009,Y -219.553,Z 1836.636,A 0.000,B 0.000,C 90.000,E1 114.463} C_DIS
LIN {X -0.059,Y -224.040,Z 1836.622,A 0.000,B 0.000,C 90.000,E1 111.897} C_DIS
LIN {X -0.110,Y -282.807,Z 1836.622,A 0.000,B 0.000,C 90.000,E1 111.897} C_DIS
LIN {X -0.154,Y -286.143,Z 1836.621,A 0.000,B 0.000,C 90.000,E1 111.844} C_DIS
LIN {X 0.009,Y -290.109,Z 1836.620,A 0.000,B 0.000,C 90.000,E1 111.589} C_DIS
LIN {X 0.069,Y -292.496,Z 1836.619,A 0.000,B 0.000,C 90.000,E1 111.354} C_DIS
LIN {X -0.079,Y -296.311,Z 1836.616,A 0.000,B 0.000,C 90.000,E1 110.844} C_DIS
LIN {X 0.096,Y -309.557,Z 1836.603,A 0.000,B 0.000,C 90.000,E1 108.489} C_DIS
LIN {X -0.104,Y -324.159,Z 1836.590,A 0.000,B 0.000,C 90.000,E1 106.260} C_DIS
LIN {X -0.052,Y -337.857,Z 1836.580,A 0.000,B 0.000,C 90.000,E1 104.356} C_DIS
LIN {X 0.106,Y -352.741,Z 1836.569,A 0.000,B 0.000,C 90.000,E1 102.479} C_DIS
LIN {X -0.202,Y -371.131,Z 1836.558,A 0.000,B 0.000,C 90.000,E1 100.489} C_DIS
LIN {X -0.144,Y -389.999,Z 1836.548,A 0.000,B 0.000,C 90.000,E1 98.624} C_DIS
LIN {X 0.189,Y -409.209,Z 1836.538,A 0.000,B 0.000,C 90.000,E1 96.891} C_DIS
LIN {X 0.031,Y -431.585,Z 1836.529,A 0.000,B 0.000,C 90.000,E1 95.163} C_DIS
LIN {X 0.184,Y -439.914,Z 1836.525,A 0.000,B 0.000,C 90.000,E1 94.531} C_DIS
LIN {X 0.036,Y -443.619,Z 1836.523,A 0.000,B 0.000,C 90.000,E1 94.131} C_DIS
LIN {X -0.209,Y -445.199,Z 1836.521,A 0.000,B 0.000,C 90.000,E1 93.898} C_DIS
LIN {X -0.041,Y -446.389,Z 1836.520,A 0.000,B 0.000,C 90.000,E1 93.612} C_DIS
LIN {X -0.090,Y -447.855,Z 1836.517,A 0.000,B 0.000,C 90.000,E1 93.094} C_DIS
LIN {X -0.157,Y -448.319,Z 1836.514,A 0.000,B 0.000,C 90.000,E1 92.579} C_DIS
LIN {X -0.212,Y -447.858,Z 1836.511,A 0.000,B 0.000,C 90.000,E1 92.064} C_DIS
LIN {X 0.198,Y -446.405,Z 1836.508,A 0.000,B 0.000,C 90.000,E1 91.489} C_DIS
LIN {X -0.052,Y -445.236,Z 1836.507,A 0.000,B 0.000,C 90.000,E1 91.260} C_DIS
LIN {X -0.009,Y -437.082,Z 1836.500,A 0.000,B 0.000,C 90.000,E1 89.943} C_DIS
LIN {X 0.056,Y -427.203,Z 1836.491,A 0.000,B 0.000,C 90.000,E1 88.339} C_DIS
LIN {X 0.074,Y -415.421,Z 1836.480,A 0.000,B 0.000,C 90.000,E1 86.445} C_DIS
LIN {X -0.102,Y -403.572,Z 1836.470,A 0.000,B 0.000,C 90.000,E1 84.546} C_DIS
LIN {X -0.126,Y -391.633,Z 1836.459,A 0.000,B 0.000,C 90.000,E1 82.591} C_DIS
LIN {X 0.076,Y -379.685,Z 1836.448,A 0.000,B 0.000,C 90.000,E1 80.566} C_DIS
LIN {X 0.120,Y -364.544,Z 1836.433,A 0.000,B 0.000,C 90.000,E1 77.937} C_DIS
LIN {X -0.133,Y -348.680,Z 1836.417,A 0.000,B 0.000,C 90.000,E1 74.991} C_DIS
LIN {X -0.115,Y -336.603,Z 1836.403,A 0.000,B 0.000,C 90.000,E1 72.543} C_DIS
LIN {X 0.121,Y -324.800,Z 1836.389,A 0.000,B 0.000,C 90.000,E1 70.007} C_DIS
LIN {X -0.049,Y -310.606,Z 1836.371,A 0.000,B 0.000,C 90.000,E1 66.847} C_DIS
LIN {X 0.107,Y -301.003,Z 1836.359,A 0.000,B 0.000,C 90.000,E1 64.537} C_DIS
LIN {X 0.012,Y -288.851,Z 1836.342,A 0.000,B 0.000,C 90.000,E1 61.563} C_DIS
LIN {X -0.047,Y -279.472,Z 1836.329,A 0.000,B 0.000,C 90.000,E1 59.203} C_DIS
LIN {X 0.032,Y -271.397,Z 1836.317,A 0.000,B 0.000,C 90.000,E1 57.120} C_DIS
LIN {X 0.028,Y -263.269,Z 1836.306,A 0.000,B 0.000,C 90.000,E1 55.022} C_DIS
LIN {X -0.088,Y -253.669,Z 1836.292,A 0.000,B 0.000,C 90.000,E1 52.557} C_DIS
LIN {X 0.047,Y -244.084,Z 1836.278,A 0.000,B 0.000,C 90.000,E1 49.989} C_DIS
LIN {X 0.089,Y -234.629,Z 1836.263,A 0.000,B 0.000,C 90.000,E1 47.391} C_DIS
LIN {X -0.053,Y -222.985,Z 1836.245,A 0.000,B 0.000,C 90.000,E1 44.028} C_DIS
LIN {X -0.093,Y -220.817,Z 1836.241,A 0.000,B 0.000,C 90.000,E1 43.380} C_DIS
LIN {X 0.044,Y -220.801,Z 1836.241,A 0.000,B 0.000,C 90.000,E1 43.338} C_DIS
LIN {X 0.043,Y -227.799,Z 1836.234,A 0.000,B 0.000,C 90.000,E1 42.081} C_DIS
LIN {X 0.126,Y -228.715,Z 1836.232,A 0.000,B 0.000,C 90.000,E1 41.676} C_DIS
LIN {X 0.015,Y -229.157,Z 1836.228,A 0.000,B 0.000,C 90.000,E1 40.943} C_DIS
LIN {X 0.061,Y -228.927,Z 1836.223,A 0.000,B 0.000,C 90.000,E1 40.172} C_DIS
LIN {X -0.040,Y -228.378,Z 1836.219,A 0.000,B 0.000,C 90.000,E1 39.439} C_DIS
LIN {X 0.078,Y -226.684,Z 1836.211,A 0.000,B 0.000,C 90.000,E1 37.890} C_DIS
LIN {X 0.034,Y -224.534,Z 1836.202,A 0.000,B 0.000,C 90.000,E1 36.377} C_DIS
LIN {X 0.061,Y -221.015,Z 1836.189,A 0.000,B 0.000,C 90.000,E1 34.072} C_DIS
LIN {X -0.102,Y -217.237,Z 1836.177,A 0.000,B 0.000,C 90.000,E1 31.799} C_DIS
LIN {X 0.091,Y -210.808,Z 1836.155,A 0.000,B 0.000,C 90.000,E1 27.847} C_DIS
LIN {X 0.067,Y -204.811,Z 1836.133,A 0.000,B 0.000,C 90.000,E1 23.898} C_DIS
LIN {X -0.091,Y -199.743,Z 1836.111,A 0.000,B 0.000,C 90.000,E1 19.939} C_DIS
LIN {X 0.075,Y -195.389,Z 1836.088,A 0.000,B 0.000,C 90.000,E1 15.843} C_DIS
LIN {X 0.024,Y -190.936,Z 1836.061,A 0.000,B 0.000,C 90.000,E1 10.950} C_DIS
LIN {X -0.067,Y -187.413,Z 1836.033,A 0.000,B 0.000,C 90.000,E1 6.024} C_DIS
LIN {X 0.045,Y -184.783,Z 1835.993,A 0.000,B 0.000,C 90.000,E1 358.682} C_DIS
LIN {X 0.005,Y -184.490,Z 1835.956,A 0.000,B 0.000,C 90.000,E1 352.008} C_DIS
LIN {X 0.007,Y -185.347,Z 1835.928,A 0.000,B 0.000,C 90.000,E1 346.992} C_DIS
LIN {X -0.030,Y -186.680,Z 1835.905,A 0.000,B 0.000,C 90.000,E1 342.834} C_DIS
LIN {X 0.046,Y -189.401,Z 1835.872,A 0.000,B 0.000,C 90.000,E1 336.997} C_DIS
LIN {X 0.113,Y -192.695,Z 1835.845,A 0.000,B 0.000,C 90.000,E1 332.025} C_DIS
LIN {X 0.085,Y -196.712,Z 1835.818,A 0.000,B 0.000,C 90.000,E1 327.120} C_DIS
LIN {X 0.002,Y -200.689,Z 1835.795,A 0.000,B 0.000,C 90.000,E1 323.084} C_DIS
LIN {X 0.017,Y -205.389,Z 1835.773,A 0.000,B 0.000,C 90.000,E1 319.057} C_DIS
LIN {X 0.020,Y -208.956,Z 1835.759,A 0.000,B 0.000,C 90.000,E1 316.662} C_DIS
LIN {X 0.002,Y -211.861,Z 1835.750,A 0.000,B 0.000,C 90.000,E1 315.081} C_DIS
LIN {X 0.019,Y -215.255,Z 1835.742,A 0.000,B 0.000,C 90.000,E1 313.500} C_DIS
LIN {X 0.080,Y -219.419,Z 1835.733,A 0.000,B 0.000,C 90.000,E1 311.919} C_DIS
LIN {X 0.053,Y -224.346,Z 1835.724,A 0.000,B 0.000,C 90.000,E1 310.378} C_DIS
LIN {X 0.115,Y -230.156,Z 1835.716,A 0.000,B 0.000,C 90.000,E1 308.830} C_DIS
LIN {X -0.075,Y -236.707,Z 1835.708,A 0.000,B 0.000,C 90.000,E1 307.363} C_DIS
LIN {X 0.027,Y -247.602,Z 1835.695,A 0.000,B 0.000,C 90.000,E1 305.105} C_DIS
LIN {X 0.104,Y -261.796,Z 1835.681,A 0.000,B 0.000,C 90.000,E1 302.546} C_DIS
LIN {X 0.025,Y -280.028,Z 1835.665,A 0.000,B 0.000,C 90.000,E1 299.745} C_DIS
LIN {X -0.117,Y -296.852,Z 1835.652,A 0.000,B 0.000,C 90.000,E1 297.385} C_DIS
LIN {X -0.069,Y -311.441,Z 1835.641,A 0.000,B 0.000,C 90.000,E1 295.387} C_DIS
LIN {X -0.140,Y -326.008,Z 1835.630,A 0.000,B 0.000,C 90.000,E1 293.462} C_DIS
LIN {X 0.102,Y -337.977,Z 1835.621,A 0.000,B 0.000,C 90.000,E1 291.844} C_DIS
LIN {X 0.078,Y -347.130,Z 1835.615,A 0.000,B 0.000,C 90.000,E1 290.610} C_DIS
LIN {X 0.045,Y -355.635,Z 1835.608,A 0.000,B 0.000,C 90.000,E1 289.396} C_DIS
LIN {X 0.059,Y -361.378,Z 1835.603,A 0.000,B 0.000,C 90.000,E1 288.489} C_DIS
LIN {X 0.135,Y -366.493,Z 1835.598,A 0.000,B 0.000,C 90.000,E1 287.583} C_DIS
LIN {X -0.179,Y -369.455,Z 1835.594,A 0.000,B 0.000,C 90.000,E1 287.040} C_DIS
LIN {X -0.122,Y -372.000,Z 1835.591,A 0.000,B 0.000,C 90.000,E1 286.441} C_DIS
LIN {X -0.038,Y -373.173,Z 1835.590,A 0.000,B 0.000,C 90.000,E1 286.134} C_DIS
LIN {X -0.059,Y -375.195,Z 1835.586,A 0.000,B 0.000,C 90.000,E1 285.552} C_DIS
LIN {X 0.031,Y -376.897,Z 1835.583,A 0.000,B 0.000,C 90.000,E1 284.954} C_DIS
LIN {X 0.131,Y -378.217,Z 1835.580,A 0.000,B 0.000,C 90.000,E1 284.356} C_DIS
LIN {X 0.148,Y -379.104,Z 1835.577,A 0.000,B 0.000,C 90.000,E1 283.772} C_DIS
LIN {X -0.106,Y -379.645,Z 1835.573,A 0.000,B 0.000,C 90.000,E1 283.231} C_DIS
LIN {X -0.074,Y -379.715,Z 1835.570,A 0.000,B 0.000,C 90.000,E1 282.647} C_DIS
LIN {X -0.038,Y -379.343,Z 1835.567,A 0.000,B 0.000,C 90.000,E1 282.063} C_DIS
LIN {X 0.000,Y -378.511,Z 1835.564,A 0.000,B 0.000,C 90.000,E1 281.478} C_DIS
LIN {X 0.037,Y -377.256,Z 1835.561,A 0.000,B 0.000,C 90.000,E1 280.894} C_DIS
LIN {X 0.066,Y -375.524,Z 1835.557,A 0.000,B 0.000,C 90.000,E1 280.310} C_DIS
LIN {X 0.031,Y -372.181,Z 1835.552,A 0.000,B 0.000,C 90.000,E1 279.443} C_DIS
LIN {X -0.075,Y -364.896,Z 1835.543,A 0.000,B 0.000,C 90.000,E1 277.701} C_DIS
LIN {X 0.156,Y -360.725,Z 1835.538,A 0.000,B 0.000,C 90.000,E1 276.777} C_DIS
LIN {X 0.035,Y -357.400,Z 1835.534,A 0.000,B 0.000,C 90.000,E1 276.201} C_DIS
LIN {X -0.101,Y -353.553,Z 1835.531,A 0.000,B 0.000,C 90.000,E1 275.625} C_DIS
LIN {X 0.092,Y -349.071,Z 1835.528,A 0.000,B 0.000,C 90.000,E1 274.992} C_DIS
LIN {X -0.088,Y -343.794,Z 1835.524,A 0.000,B 0.000,C 90.000,E1 274.416} C_DIS
LIN {X 0.165,Y -338.003,Z 1835.521,A 0.000,B 0.000,C 90.000,E1 273.784} C_DIS
LIN {X 0.009,Y -332.041,Z 1835.518,A 0.000,B 0.000,C 90.000,E1 273.269} C_DIS
LIN {X 0.103,Y -325.805,Z 1835.515,A 0.000,B 0.000,C 90.000,E1 272.751} C_DIS
LIN {X 0.097,Y -319.226,Z 1835.513,A 0.000,B 0.000,C 90.000,E1 272.293} C_DIS
LIN {X 0.100,Y -312.636,Z 1835.511,A 0.000,B 0.000,C 90.000,E1 271.892} C_DIS
LIN {X 0.036,Y -305.630,Z 1835.509,A 0.000,B 0.000,C 90.000,E1 271.547} C_DIS
LIN {X -0.049,Y -298.045,Z 1835.507,A 0.000,B 0.000,C 90.000,E1 271.260} C_DIS
LIN {X -0.099,Y -290.171,Z 1835.506,A 0.000,B 0.000,C 90.000,E1 271.031} C_DIS
LIN {X -0.007,Y -278.810,Z 1835.504,A 0.000,B 0.000,C 90.000,E1 270.745} C_DIS
LIN {X 0.104,Y -249.579,Z 1835.501,A 0.000,B 0.000,C 90.000,E1 270.172} C_DIS
LIN {X 0.026,Y -240.732,Z 1835.500,A 0.000,B 0.000,C 90.000,E1 270.057} C_DIS
LIN {X 0.064,Y -235.202,Z 1835.500,A 0.000,B 0.000,C 90.000,E1 270.000} C_DIS
LIN {X -0.002,Y -229.968,Z 1835.500,A 0.000,B 0.000,C 90.000,E1 270.000} C_DIS
LIN {X -0.027,Y -181.559,Z 1835.500,A 0.000,B 0.000,C 90.000,E1 270.000} C_DIS
LIN {X -0.043,Y -180.830,Z 1835.472,A 0.000,B 0.000,C 90.000,E1 264.894} C_DIS
LIN {X 0.037,Y -178.936,Z 1835.443,A 0.000,B 0.000,C 90.000,E1 259.803} C_DIS
LIN {X -0.095,Y -175.985,Z 1835.415,A 0.000,B 0.000,C 90.000,E1 254.755} C_DIS
LIN {X 0.020,Y -175.482,Z 1835.410,A 0.000,B 0.000,C 90.000,E1 253.866} C_DIS
LIN {X 0.076,Y -172.228,Z 1835.387,A 0.000,B 0.000,C 90.000,E1 249.571} C_DIS
LIN {X 0.053,Y -171.705,Z 1835.382,A 0.000,B 0.000,C 90.000,E1 248.720} C_DIS
LIN {X -0.021,Y -167.300,Z 1835.353,A 0.000,B 0.000,C 90.000,E1 243.563} C_DIS
LIN {X -0.015,Y -166.677,Z 1835.348,A 0.000,B 0.000,C 90.000,E1 242.692} C_DIS
LIN {X -0.024,Y -162.660,Z 1835.324,A 0.000,B 0.000,C 90.000,E1 238.329} C_DIS
LIN {X 0.038,Y -161.349,Z 1835.314,A 0.000,B 0.000,C 90.000,E1 236.548} C_DIS
LIN {X -0.017,Y -157.343,Z 1835.290,A 0.000,B 0.000,C 90.000,E1 232.145} C_DIS
LIN {X 0.013,Y -155.329,Z 1835.275,A 0.000,B 0.000,C 90.000,E1 229.461} C_DIS
LIN {X -0.057,Y -151.680,Z 1835.250,A 0.000,B 0.000,C 90.000,E1 225.000} C_DIS
LIN {X -0.009,Y -150.544,Z 1835.240,A 0.000,B 0.000,C 90.000,E1 223.176} C_DIS
LIN {X 0.024,Y -147.270,Z 1835.215,A 0.000,B 0.000,C 90.000,E1 218.624} C_DIS
LIN {X -0.003,Y -145.298,Z 1835.194,A 0.000,B 0.000,C 90.000,E1 214.978} C_DIS
LIN {X -0.011,Y -142.393,Z 1835.164,A 0.000,B 0.000,C 90.000,E1 209.461} C_DIS
LIN {X 0.036,Y -141.373,Z 1835.148,A 0.000,B 0.000,C 90.000,E1 206.668} C_DIS
LIN {X 0.013,Y -139.346,Z 1835.112,A 0.000,B 0.000,C 90.000,E1 200.174} C_DIS
LIN {X -0.045,Y -138.782,Z 1835.097,A 0.000,B 0.000,C 90.000,E1 197.402} C_DIS
LIN {X 0.014,Y -138.343,Z 1835.055,A 0.000,B 0.000,C 90.000,E1 189.905} C_DIS
LIN {X 0.034,Y -139.392,Z 1835.008,A 0.000,B 0.000,C 90.000,E1 181.489} C_DIS
LIN {X -0.052,Y -141.291,Z 1834.972,A 0.000,B 0.000,C 90.000,E1 175.008} C_DIS
LIN {X 0.046,Y -142.653,Z 1834.957,A 0.000,B 0.000,C 90.000,E1 172.186} C_DIS
LIN {X -0.004,Y -144.993,Z 1834.931,A 0.000,B 0.000,C 90.000,E1 167.589} C_DIS
LIN {X -0.014,Y -147.621,Z 1834.911,A 0.000,B 0.000,C 90.000,E1 163.921} C_DIS
LIN {X 0.064,Y -150.246,Z 1834.890,A 0.000,B 0.000,C 90.000,E1 160.242} C_DIS
LIN {X -0.062,Y -153.642,Z 1834.870,A 0.000,B 0.000,C 90.000,E1 156.666} C_DIS
LIN {X -0.005,Y -157.056,Z 1834.850,A 0.000,B 0.000,C 90.000,E1 153.050} C_DIS
LIN {X -0.007,Y -161.186,Z 1834.830,A 0.000,B 0.000,C 90.000,E1 149.488} C_DIS
LIN {X 0.023,Y -163.279,Z 1834.821,A 0.000,B 0.000,C 90.000,E1 147.709} C_DIS
LIN {X 0.035,Y -167.722,Z 1834.801,A 0.000,B 0.000,C 90.000,E1 144.196} C_DIS
LIN {X -0.053,Y -171.542,Z 1834.787,A 0.000,B 0.000,C 90.000,E1 141.618} C_DIS
LIN {X -0.011,Y -176.483,Z 1834.768,A 0.000,B 0.000,C 90.000,E1 138.162} C_DIS
LIN {X -0.011,Y -180.780,Z 1834.753,A 0.000,B 0.000,C 90.000,E1 135.607} C_DIS
LIN {X -0.024,Y -186.187,Z 1834.735,A 0.000,B 0.000,C 90.000,E1 132.243} C_DIS
LIN {X 0.040,Y -190.825,Z 1834.721,A 0.000,B 0.000,C 90.000,E1 129.725} C_DIS
LIN {X -0.041,Y -196.584,Z 1834.703,A 0.000,B 0.000,C 90.000,E1 126.457} C_DIS
LIN {X 0.043,Y -201.351,Z 1834.689,A 0.000,B 0.000,C 90.000,E1 123.992} C_DIS
LIN {X -0.029,Y -207.329,Z 1834.671,A 0.000,B 0.000,C 90.000,E1 120.797} C_DIS
LIN {X -0.030,Y -210.577,Z 1834.662,A 0.000,B 0.000,C 90.000,E1 119.205} C_DIS
LIN {X -0.030,Y -216.386,Z 1834.645,A 0.000,B 0.000,C 90.000,E1 116.052} C_DIS
LIN {X 0.077,Y -219.516,Z 1834.636,A 0.000,B 0.000,C 90.000,E1 114.463} C_DIS
LIN {X -0.058,Y -224.039,Z 1834.622,A 0.000,B 0.000,C 90.000,E1 111.897} C_DIS
LIN {X -0.102,Y -282.764,Z 1834.622,A 0.000,B 0.000,C 90.000,E1 111.897} C_DIS
LIN {X -0.046,Y -285.501,Z 1834.621,A 0.000,B 0.000,C 90.000,E1 111.844} C_DIS
LIN {X 0.121,Y -289.831,Z 1834.620,A 0.000,B 0.000,C 90.000,E1 111.589} C_DIS
LIN {X -0.090,Y -292.295,Z 1834.619,A 0.000,B 0.000,C 90.000,E1 111.408} C_DIS
LIN {X 0.002,Y -296.106,Z 1834.616,A 0.000,B 0.000,C 90.000,E1 110.865} C_DIS
LIN {X -0.007,Y -309.342,Z 1834.603,A 0.000,B 0.000,C 90.000,E1 108.544} C_DIS
LIN {X 0.091,Y -323.922,Z 1834.590,A 0.000,B 0.000,C 90.000,E1 106.260} C_DIS
LIN {X 0.147,Y -337.599,Z 1834.580,A 0.000,B 0.000,C 90.000,E1 104.356} C_DIS
LIN {X -0.036,Y -352.462,Z 1834.570,A 0.000,B 0.000,C 90.000,E1 102.535} C_DIS
LIN {X -0.009,Y -370.844,Z 1834.558,A 0.000,B 0.000,C 90.000,E1 100.489} C_DIS
LIN {X 0.041,Y -389.705,Z 1834.548,A 0.000,B 0.000,C 90.000,E1 98.624} C_DIS
LIN {X -0.040,Y -408.911,Z 1834.539,A 0.000,B 0.000,C 90.000,E1 96.947} C_DIS
LIN {X 0.199,Y -431.281,Z 1834.529,A 0.000,B 0.000,C 90.000,E1 95.163} C_DIS
LIN {X -0.090,Y -439.659,Z 1834.525,A 0.000,B 0.000,C 90.000,E1 94.588} C_DIS
LIN {X -0.198,Y -443.422,Z 1834.523,A 0.000,B 0.000,C 90.000,E1 94.188} C_DIS
LIN {X 0.000,Y -445.048,Z 1834.522,A 0.000,B 0.000,C 90.000,E1 93.898} C_DIS
LIN {X 0.168,Y -446.273,Z 1834.520,A 0.000,B 0.000,C 90.000,E1 93.612} C_DIS
LIN {X 0.118,Y -447.793,Z 1834.517,A 0.000,B 0.000,C 90.000,E1 93.094} C_DIS
LIN {X 0.052,Y -448.305,Z 1834.514,A 0.000,B 0.000,C 90.000,E1 92.579} C_DIS
LIN {X -0.004,Y -447.889,Z 1834.511,A 0.000,B 0.000,C 90.000,E1 92.064} C_DIS
LIN {X -0.041,Y -446.490,Z 1834.509,A 0.000,B 0.000,C 90.000,E1 91.547} C_DIS
LIN {X 0.155,Y -445.353,Z 1834.507,A 0.000,B 0.000,C 90.000,E1 91.260} C_DIS
LIN {X -0.160,Y -440.536,Z 1834.503,A 0.000,B 0.000,C 90.000,E1 90.516} C_DIS
LIN {X 0.115,Y -429.009,Z 1834.492,A 0.000,B 0.000,C 90.000,E1 88.625} C_DIS
LIN {X 0.176,Y -417.248,Z 1834.482,A 0.000,B 0.000,C 90.000,E1 86.731} C_DIS
LIN {X -0.003,Y -405.429,Z 1834.471,A 0.000,B 0.000,C 90.000,E1 84.837} C_DIS
LIN {X 0.057,Y -393.497,Z 1834.460,A 0.000,B 0.000,C 90.000,E1 82.875} C_DIS
LIN {X -0.079,Y -381.550,Z 1834.449,A 0.000,B 0.000,C 90.000,E1 80.905} C_DIS
LIN {X -0.026,Y -367.999,Z 1834.437,A 0.000,B 0.000,C 90.000,E1 78.578} C_DIS
LIN {X 0.118,Y -350.358,Z 1834.418,A 0.000,B 0.000,C 90.000,E1 75.283} C_DIS
LIN {X 0.073,Y -338.227,Z 1834.405,A 0.000,B 0.000,C 90.000,E1 72.851} C_DIS
LIN {X 0.030,Y -326.381,Z 1834.391,A 0.000,B 0.000,C 90.000,E1 70.369} C_DIS
LIN {X 0.082,Y -312.107,Z 1834.373,A 0.000,B 0.000,C 90.000,E1 67.177} C_DIS
LIN {X -0.019,Y -302.488,Z 1834.361,A 0.000,B 0.000,C 90.000,E1 64.921} C_DIS
LIN {X -0.066,Y -290.285,Z 1834.344,A 0.000,B 0.000,C 90.000,E1 61.948} C_DIS
LIN {X 0.152,Y -280.926,Z 1834.331,A 0.000,B 0.000,C 90.000,E1 59.537} C_DIS
LIN {X -0.035,Y -271.510,Z 1834.318,A 0.000,B 0.000,C 90.000,E1 57.168} C_DIS
LIN {X 0.036,Y -263.387,Z 1834.306,A 0.000,B 0.000,C 90.000,E1 55.055} C_DIS
LIN {X 0.067,Y -253.784,Z 1834.292,A 0.000,B 0.000,C 90.000,E1 52.557} C_DIS
LIN {X 0.011,Y -244.199,Z 1834.278,A 0.000,B 0.000,C 90.000,E1 50.033} C_DIS
LIN {X -0.094,Y -234.741,Z 1834.264,A 0.000,B 0.000,C 90.000,E1 47.472} C_DIS
LIN {X -0.037,Y -227.861,Z 1834.253,A 0.000,B 0.000,C 90.000,E1 45.486} C_DIS
LIN {X -0.060,Y -227.853,Z 1834.253,A 0.000,B 0.000,C 90.000,E1 45.486} C_DIS
LIN {X 0.006,Y -233.407,Z 1834.247,A 0.000,B 0.000,C 90.000,E1 44.433} C_DIS
LIN {X 0.113,Y -234.931,Z 1834.245,A 0.000,B 0.000,C 90.000,E1 44.028} C_DIS
LIN {X 0.017,Y -235.652,Z 1834.241,A 0.000,B 0.000,C 90.000,E1 43.299} C_DIS
LIN {X 0.103,Y -235.487,Z 1834.236,A 0.000,B 0.000,C 90.000,E1 42.528} C_DIS
LIN {X -0.138,Y -234.922,Z 1834.232,A 0.000,B 0.000,C 90.000,E1 41.838} C_DIS
LIN {X 0.035,Y -233.157,Z 1834.224,A 0.000,B 0.000,C 90.000,E1 40.297} C_DIS
LIN {X -0.112,Y -231.000,Z 1834.216,A 0.000,B 0.000,C 90.000,E1 38.830} C_DIS
LIN {X 0.039,Y -228.523,Z 1834.207,A 0.000,B 0.000,C 90.000,E1 37.282} C_DIS
LIN {X -0.048,Y -224.501,Z 1834.194,A 0.000,B 0.000,C 90.000,E1 35.025} C_DIS
LIN {X 0.038,Y -220.448,Z 1834.182,A 0.000,B 0.000,C 90.000,E1 32.704} C_DIS
LIN {X 0.006,Y -214.828,Z 1834.165,A 0.000,B 0.000,C 90.000,E1 29.617} C_DIS
LIN {X -0.080,Y -208.193,Z 1834.143,A 0.000,B 0.000,C 90.000,E1 25.720} C_DIS
LIN {X 0.022,Y -203.382,Z 1834.125,A 0.000,B 0.000,C 90.000,E1 22.514} C_DIS
LIN {X 0.050,Y -198.287,Z 1834.103,A 0.000,B 0.000,C 90.000,E1 18.489} C_DIS
LIN {X 0.058,Y -193.888,Z 1834.080,A 0.000,B 0.000,C 90.000,E1 14.426} C_DIS
LIN {X -0.079,Y -190.049,Z 1834.057,A 0.000,B 0.000,C 90.000,E1 10.366} C_DIS
LIN {X -0.042,Y -186.672,Z 1834.030,A 0.000,B 0.000,C 90.000,E1 5.391} C_DIS
LIN {X -0.062,Y -184.259,Z 1833.988,A 0.000,B 0.000,C 90.000,E1 357.879} C_DIS
LIN {X 0.080,Y -184.195,Z 1833.951,A 0.000,B 0.000,C 90.000,E1 351.141} C_DIS
LIN {X 0.098,Y -185.464,Z 1833.918,A 0.000,B 0.000,C 90.000,E1 345.283} C_DIS
LIN {X -0.009,Y -187.353,Z 1833.891,A 0.000,B 0.000,C 90.000,E1 340.315} C_DIS
LIN {X -0.090,Y -190.664,Z 1833.858,A 0.000,B 0.000,C 90.000,E1 334.537} C_DIS
LIN {X -0.048,Y -194.351,Z 1833.831,A 0.000,B 0.000,C 90.000,E1 329.587} C_DIS
LIN {X 0.078,Y -197.989,Z 1833.808,A 0.000,B 0.000,C 90.000,E1 325.468} C_DIS
LIN {X -0.049,Y -202.263,Z 1833.786,A 0.000,B 0.000,C 90.000,E1 321.457} C_DIS
LIN {X -0.038,Y -206.393,Z 1833.768,A 0.000,B 0.000,C 90.000,E1 318.243} C_DIS
LIN {X 0.121,Y -210.321,Z 1833.755,A 0.000,B 0.000,C 90.000,E1 315.810} C_DIS
LIN {X -0.033,Y -213.535,Z 1833.746,A 0.000,B 0.000,C 90.000,E1 314.271} C_DIS
LIN {X 0.003,Y -217.345,Z 1833.737,A 0.000,B 0.000,C 90.000,E1 312.690} C_DIS
LIN {X -0.050,Y -221.944,Z 1833.729,A 0.000,B 0.000,C 90.000,E1 311.148} C_DIS
LIN {X 0.124,Y -227.351,Z 1833.720,A 0.000,B 0.000,C 90.000,E1 309.564} C_DIS
LIN {X -0.099,Y -233.594,Z 1833.712,A 0.000,B 0.000,C 90.000,E1 308.096} C_DIS
LIN {X 0.085,Y -244.134,Z 1833.699,A 0.000,B 0.000,C 90.000,E1 305.804} C_DIS
LIN {X -0.016,Y -253.847,Z 1833.689,A 0.000,B 0.000,C 90.000,E1 303.992} C_DIS
LIN {X -0.117,Y -264.370,Z 1833.679,A 0.000,B 0.000,C 90.000,E1 302.212} C_DIS
LIN {X -0.142,Y -282.815,Z 1833.663,A 0.000,B 0.000,C 90.000,E1 299.411} C_DIS
LIN {X 0.043,Y -297.319,Z 1833.652,A 0.000,B 0.000,C 90.000,E1 297.334} C_DIS
LIN {X 0.114,Y -311.959,Z 1833.641,A 0.000,B 0.000,C 90.000,E1 295.335} C_DIS
LIN {X 0.197,Y -326.614,Z 1833.630,A 0.000,B 0.000,C 90.000,E1 293.387} C_DIS
LIN {X 0.015,Y -338.639,Z 1833.621,A 0.000,B 0.000,C 90.000,E1 291.844} C_DIS
LIN {X -0.002,Y -347.791,Z 1833.615,A 0.000,B 0.000,C 90.000,E1 290.610} C_DIS
LIN {X 0.053,Y -354.235,Z 1833.609,A 0.000,B 0.000,C 90.000,E1 289.685} C_DIS
LIN {X 0.056,Y -360.182,Z 1833.604,A 0.000,B 0.000,C 90.000,E1 288.779} C_DIS
LIN {X 0.111,Y -365.550,Z 1833.599,A 0.000,B 0.000,C 90.000,E1 287.873} C_DIS
LIN {X 0.142,Y -368.707,Z 1833.596,A 0.000,B 0.000,C 90.000,E1 287.275} C_DIS
LIN {X 0.194,Y -371.460,Z 1833.593,A 0.000,B 0.000,C 90.000,E1 286.677} C_DIS
LIN {X -0.093,Y -373.796,Z 1833.590,A 0.000,B 0.000,C 90.000,E1 286.134} C_DIS
LIN {X -0.110,Y -375.804,Z 1833.586,A 0.000,B 0.000,C 90.000,E1 285.552} C_DIS
LIN {X -0.017,Y -377.465,Z 1833.583,A 0.000,B 0.000,C 90.000,E1 284.954} C_DIS
LIN {X 0.087,Y -378.757,Z 1833.580,A 0.000,B 0.000,C 90.000,E1 284.356} C_DIS
LIN {X 0.107,Y -379.651,Z 1833.577,A 0.000,B 0.000,C 90.000,E1 283.772} C_DIS
LIN {X -0.145,Y -380.155,Z 1833.573,A 0.000,B 0.000,C 90.000,E1 283.231} C_DIS
LIN {X -0.109,Y -380.210,Z 1833.570,A 0.000,B 0.000,C 90.000,E1 282.647} C_DIS
LIN {X -0.069,Y -379.825,Z 1833.567,A 0.000,B 0.000,C 90.000,E1 282.063} C_DIS
LIN {X -0.028,Y -378.987,Z 1833.564,A 0.000,B 0.000,C 90.000,E1 281.478} C_DIS
LIN {X 0.011,Y -377.688,Z 1833.561,A 0.000,B 0.000,C 90.000,E1 280.894} C_DIS
LIN {X 0.044,Y -375.936,Z 1833.557,A 0.000,B 0.000,C 90.000,E1 280.310} C_DIS
LIN {X 0.013,Y -372.608,Z 1833.552,A 0.000,B 0.000,C 90.000,E1 279.443} C_DIS
LIN {X -0.086,Y -365.259,Z 1833.543,A 0.000,B 0.000,C 90.000,E1 277.701} C_DIS
LIN {X 0.149,Y -360.983,Z 1833.538,A 0.000,B 0.000,C 90.000,E1 276.777} C_DIS
LIN {X -0.019,Y -355.757,Z 1833.533,A 0.000,B 0.000,C 90.000,E1 275.910} C_DIS
LIN {X 0.184,Y -351.594,Z 1833.530,A 0.000,B 0.000,C 90.000,E1 275.277} C_DIS
LIN {X 0.014,Y -346.675,Z 1833.526,A 0.000,B 0.000,C 90.000,E1 274.702} C_DIS
LIN {X -0.149,Y -341.148,Z 1833.523,A 0.000,B 0.000,C 90.000,E1 274.131} C_DIS
LIN {X -0.100,Y -335.187,Z 1833.520,A 0.000,B 0.000,C 90.000,E1 273.555} C_DIS
LIN {X -0.127,Y -329.044,Z 1833.517,A 0.000,B 0.000,C 90.000,E1 273.037} C_DIS
LIN {X 0.076,Y -322.699,Z 1833.514,A 0.000,B 0.000,C 90.000,E1 272.522} C_DIS
LIN {X -0.083,Y -316.083,Z 1833.512,A 0.000,B 0.000,C 90.000,E1 272.121} C_DIS
LIN {X 0.061,Y -309.339,Z 1833.510,A 0.000,B 0.000,C 90.000,E1 271.718} C_DIS
LIN {X -0.142,Y -302.108,Z 1833.508,A 0.000,B 0.000,C 90.000,E1 271.432} C_DIS
LIN {X -0.034,Y -294.436,Z 1833.506,A 0.000,B 0.000,C 90.000,E1 271.146} C_DIS
LIN {X -0.114,Y -282.974,Z 1833.505,A 0.000,B 0.000,C 90.000,E1 270.859} C_DIS
LIN {X 0.113,Y -268.087,Z 1833.503,A 0.000,B 0.000,C 90.000,E1 270.516} C_DIS
LIN {X -0.095,Y -250.380,Z 1833.501,A 0.000,B 0.000,C 90.000,E1 270.229} C_DIS
LIN {X 0.076,Y -241.473,Z 1833.500,A 0.000,B 0.000,C 90.000,E1 270.057} C_DIS
LIN {X 0.051,Y -231.860,Z 1833.500,A 0.000,B 0.000,C 90.000,E1 270.000} C_DIS
LIN {X 0.005,Y -181.561,Z 1833.500,A 0.000,B 0.000,C 90.000,E1 270.000} C_DIS
LIN {X -0.066,Y -180.829,Z 1833.472,A 0.000,B 0.000,C 90.000,E1 264.894} C_DIS
LIN {X 0.014,Y -178.934,Z 1833.443,A 0.000,B 0.000,C 90.000,E1 259.803} C_DIS
LIN {X 0.052,Y -175.982,Z 1833.415,A 0.000,B 0.000,C 90.000,E1 254.700} C_DIS
LIN {X -0.004,Y -175.475,Z 1833.410,A 0.000,B 0.000,C 90.000,E1 253.866} C_DIS
LIN {X 0.053,Y -172.223,Z 1833.387,A 0.000,B 0.000,C 90.000,E1 249.571} C_DIS
LIN {X 0.031,Y -171.700,Z 1833.382,A 0.000,B 0.000,C 90.000,E1 248.720} C_DIS
LIN {X -0.043,Y -167.294,Z 1833.353,A 0.000,B 0.000,C 90.000,E1 243.563} C_DIS
LIN {X 0.039,Y -166.671,Z 1833.348,A 0.000,B 0.000,C 90.000,E1 242.666} C_DIS
LIN {X -0.046,Y -162.654,Z 1833.324,A 0.000,B 0.000,C 90.000,E1 238.329} C_DIS
LIN {X 0.016,Y -161.343,Z 1833.314,A 0.000,B 0.000,C 90.000,E1 236.548} C_DIS
LIN {X 0.059,Y -157.337,Z 1833.290,A 0.000,B 0.000,C 90.000,E1 232.110} C_DIS
LIN {X -0.008,Y -155.321,Z 1833.275,A 0.000,B 0.000,C 90.000,E1 229.461} C_DIS
LIN {X -0.078,Y -151.674,Z 1833.250,A 0.000,B 0.000,C 90.000,E1 225.000} C_DIS
LIN {X -0.029,Y -150.540,Z 1833.240,A 0.000,B 0.000,C 90.000,E1 223.176} C_DIS
LIN {X 0.004,Y -147.265,Z 1833.215,A 0.000,B 0.000,C 90.000,E1 218.624} C_DIS
LIN {X -0.024,Y -145.292,Z 1833.194,A 0.000,B 0.000,C 90.000,E1 214.978} C_DIS
LIN {X -0.031,Y -142.390,Z 1833.164,A 0.000,B 0.000,C 90.000,E1 209.461} C_DIS
LIN {X 0.016,Y -141.369,Z 1833.148,A 0.000,B 0.000,C 90.000,E1 206.668} C_DIS
LIN {X -0.007,Y -139.346,Z 1833.112,A 0.000,B 0.000,C 90.000,E1 200.174} C_DIS
LIN {X -0.002,Y -139.016,Z 1833.102,A 0.000,B 0.000,C 90.000,E1 198.308} C_DIS
LIN {X -0.006,Y -138.342,Z 1833.055,A 0.000,B 0.000,C 90.000,E1 189.905} C_DIS
LIN {X 0.014,Y -139.393,Z 1833.008,A 0.000,B 0.000,C 90.000,E1 181.489} C_DIS
LIN {X 0.068,Y -141.294,Z 1832.972,A 0.000,B 0.000,C 90.000,E1 174.951} C_DIS
LIN {X 0.026,Y -142.656,Z 1832.957,A 0.000,B 0.000,C 90.000,E1 172.186} C_DIS
LIN {X -0.025,Y -144.999,Z 1832.931,A 0.000,B 0.000,C 90.000,E1 167.589} C_DIS
LIN {X -0.035,Y -147.626,Z 1832.911,A 0.000,B 0.000,C 90.000,E1 163.921} C_DIS
LIN {X 0.043,Y -150.253,Z 1832.890,A 0.000,B 0.000,C 90.000,E1 160.242} C_DIS
LIN {X 0.058,Y -153.650,Z 1832.870,A 0.000,B 0.000,C 90.000,E1 156.613} C_DIS
LIN {X -0.026,Y -157.065,Z 1832.850,A 0.000,B 0.000,C 90.000,E1 153.050} C_DIS
LIN {X 0.053,Y -161.196,Z 1832.830,A 0.000,B 0.000,C 90.000,E1 149.459} C_DIS
LIN {X 0.002,Y -163.288,Z 1832.821,A 0.000,B 0.000,C 90.000,E1 147.709} C_DIS
LIN {X 0.012,Y -167.733,Z 1832.801,A 0.000,B 0.000,C 90.000,E1 144.196} C_DIS
LIN {X -0.076,Y -171.551,Z 1832.787,A 0.000,B 0.000,C 90.000,E1 141.618} C_DIS
LIN {X -0.034,Y -176.495,Z 1832.767,A 0.000,B 0.000,C 90.000,E1 138.162} C_DIS
LIN {X 0.091,Y -180.793,Z 1832.753,A 0.000,B 0.000,C 90.000,E1 135.567} C_DIS
LIN {X -0.048,Y -186.200,Z 1832.735,A 0.000,B 0.000,C 90.000,E1 132.243} C_DIS
LIN {X 0.016,Y -190.837,Z 1832.721,A 0.000,B 0.000,C 90.000,E1 129.725} C_DIS
LIN {X 0.050,Y -196.597,Z 1832.702,A 0.000,B 0.000,C 90.000,E1 126.423} C_DIS
LIN {X 0.018,Y -201.364,Z 1832.689,A 0.000,B 0.000,C 90.000,E1 123.992} C_DIS
LIN {X -0.055,Y -207.342,Z 1832.671,A 0.000,B 0.000,C 90.000,E1 120.797} C_DIS
LIN {X -0.056,Y -210.588,Z 1832.662,A 0.000,B 0.000,C 90.000,E1 119.205} C_DIS
LIN {X 0.039,Y -216.400,Z 1832.645,A 0.000,B 0.000,C 90.000,E1 116.027} C_DIS
LIN {X 0.051,Y -219.528,Z 1832.636,A 0.000,B 0.000,C 90.000,E1 114.463} C_DIS
LIN {X -0.056,Y -224.038,Z 1832.622,A 0.000,B 0.000,C 90.000,E1 111.897} C_DIS
LIN {X -0.106,Y -283.310,Z 1832.622,A 0.000,B 0.000,C 90.000,E1 111.897} C_DIS
LIN {X -0.078,Y -285.768,Z 1832.621,A 0.000,B 0.000,C 90.000,E1 111.844} C_DIS
LIN {X 0.087,Y -289.933,Z 1832.620,A 0.000,B 0.000,C 90.000,E1 111.589} C_DIS
LIN {X -0.124,Y -292.364,Z 1832.619,A 0.000,B 0.000,C 90.000,E1 111.408} C_DIS
LIN {X 0.043,Y -296.177,Z 1832.616,A 0.000,B 0.000,C 90.000,E1 110.844} C_DIS
LIN {X -0.073,Y -309.415,Z 1832.603,A 0.000,B 0.000,C 90.000,E1 108.544} C_DIS
LIN {X 0.023,Y -324.003,Z 1832.590,A 0.000,B 0.000,C 90.000,E1 106.260} C_DIS
LIN {X 0.077,Y -337.688,Z 1832.580,A 0.000,B 0.000,C 90.000,E1 104.356} C_DIS
LIN {X -0.106,Y -352.557,Z 1832.570,A 0.000,B 0.000,C 90.000,E1 102.535} C_DIS
LIN {X -0.077,Y -370.943,Z 1832.558,A 0.000,B 0.000,C 90.000,E1 100.489} C_DIS
LIN {X -0.024,Y -389.807,Z 1832.548,A 0.000,B 0.000,C 90.000,E1 98.624} C_DIS
LIN {X -0.102,Y -409.014,Z 1832.539,A 0.000,B 0.000,C 90.000,E1 96.947} C_DIS
LIN {X 0.139,Y -431.386,Z 1832.529,A 0.000,B 0.000,C 90.000,E1 95.163} C_DIS
LIN {X -0.149,Y -439.745,Z 1832.525,A 0.000,B 0.000,C 90.000,E1 94.588} C_DIS
LIN {X 0.169,Y -443.483,Z 1832.523,A 0.000,B 0.000,C 90.000,E1 94.131} C_DIS
LIN {X -0.076,Y -445.090,Z 1832.522,A 0.000,B 0.000,C 90.000,E1 93.898} C_DIS
LIN {X 0.093,Y -446.301,Z 1832.520,A 0.000,B 0.000,C 90.000,E1 93.612} C_DIS
LIN {X 0.043,Y -447.800,Z 1832.517,A 0.000,B 0.000,C 90.000,E1 93.094} C_DIS
LIN {X -0.024,Y -448.292,Z 1832.514,A 0.000,B 0.000,C 90.000,E1 92.579} C_DIS
LIN {X -0.079,Y -447.859,Z 1832.511,A 0.000,B 0.000,C 90.000,E1 92.064} C_DIS
LIN {X -0.116,Y -446.437,Z 1832.509,A 0.000,B 0.000,C 90.000,E1 91.547} C_DIS
LIN {X 0.080,Y -445.287,Z 1832.507,A 0.000,B 0.000,C 90.000,E1 91.260} C_DIS
LIN {X -0.056,Y -438.802,Z 1832.501,A 0.000,B 0.000,C 90.000,E1 90.229} C_DIS
LIN {X 0.184,Y -427.271,Z 1832.491,A 0.000,B 0.000,C 90.000,E1 88.339} C_DIS
LIN {X 0.200,Y -415.492,Z 1832.480,A 0.000,B 0.000,C 90.000,E1 86.445} C_DIS
LIN {X 0.022,Y -403.642,Z 1832.470,A 0.000,B 0.000,C 90.000,E1 84.546} C_DIS
LIN {X -0.005,Y -391.706,Z 1832.459,A 0.000,B 0.000,C 90.000,E1 82.591} C_DIS
LIN {X -0.178,Y -379.754,Z 1832.448,A 0.000,B 0.000,C 90.000,E1 80.622} C_DIS
LIN {X -0.121,Y -364.609,Z 1832.433,A 0.000,B 0.000,C 90.000,E1 77.993} C_DIS
LIN {X 0.005,Y -347.205,Z 1832.415,A 0.000,B 0.000,C 90.000,E1 74.685} C_DIS
LIN {X -0.010,Y -335.167,Z 1832.401,A 0.000,B 0.000,C 90.000,E1 72.236} C_DIS
LIN {X -0.114,Y -323.386,Z 1832.387,A 0.000,B 0.000,C 90.000,E1 69.752} C_DIS
LIN {X -0.023,Y -309.264,Z 1832.370,A 0.000,B 0.000,C 90.000,E1 66.538} C_DIS
LIN {X -0.175,Y -299.665,Z 1832.357,A 0.000,B 0.000,C 90.000,E1 64.280} C_DIS
LIN {X -0.038,Y -287.558,Z 1832.340,A 0.000,B 0.000,C 90.000,E1 61.257} C_DIS
LIN {X 0.008,Y -278.172,Z 1832.327,A 0.000,B 0.000,C 90.000,E1 58.869} C_DIS
LIN {X 0.139,Y -268.731,Z 1832.314,A 0.000,B 0.000,C 90.000,E1 56.421} C_DIS
LIN {X -0.065,Y -260.563,Z 1832.302,A 0.000,B 0.000,C 90.000,E1 54.356} C_DIS
LIN {X 0.036,Y -252.346,Z 1832.290,A 0.000,B 0.000,C 90.000,E1 52.190} C_DIS
LIN {X -0.053,Y -242.756,Z 1832.276,A 0.000,B 0.000,C 90.000,E1 49.666} C_DIS
LIN {X -0.107,Y -235.002,Z 1832.264,A 0.000,B 0.000,C 90.000,E1 47.553} C_DIS
LIN {X -0.131,Y -234.988,Z 1832.264,A 0.000,B 0.000,C 90.000,E1 47.553} C_DIS
LIN {X 0.063,Y -241.112,Z 1832.257,A 0.000,B 0.000,C 90.000,E1 46.296} C_DIS
LIN {X 0.005,Y -242.230,Z 1832.253,A 0.000,B 0.000,C 90.000,E1 45.567} C_DIS
LIN {X -0.043,Y -242.151,Z 1832.249,A 0.000,B 0.000,C 90.000,E1 44.838} C_DIS
LIN {X -0.083,Y -241.594,Z 1832.245,A 0.000,B 0.000,C 90.000,E1 44.109} C_DIS
LIN {X 0.051,Y -240.785,Z 1832.241,A 0.000,B 0.000,C 90.000,E1 43.338} C_DIS
LIN {X 0.130,Y -238.706,Z 1832.233,A 0.000,B 0.000,C 90.000,E1 41.838} C_DIS
LIN {X 0.022,Y -236.230,Z 1832.224,A 0.000,B 0.000,C 90.000,E1 40.378} C_DIS
LIN {X -0.006,Y -232.216,Z 1832.212,A 0.000,B 0.000,C 90.000,E1 38.141} C_DIS
LIN {X -0.027,Y -227.819,Z 1832.199,A 0.000,B 0.000,C 90.000,E1 35.884} C_DIS
LIN {X -0.009,Y -221.953,Z 1832.182,A 0.000,B 0.000,C 90.000,E1 32.832} C_DIS
LIN {X -0.006,Y -215.975,Z 1832.165,A 0.000,B 0.000,C 90.000,E1 29.745} C_DIS
LIN {X -0.060,Y -208.941,Z 1832.144,A 0.000,B 0.000,C 90.000,E1 25.848} C_DIS
LIN {X 0.061,Y -203.829,Z 1832.126,A 0.000,B 0.000,C 90.000,E1 22.642} C_DIS
LIN {X -0.024,Y -198.401,Z 1832.104,A 0.000,B 0.000,C 90.000,E1 18.652} C_DIS
LIN {X -0.024,Y -193.686,Z 1832.081,A 0.000,B 0.000,C 90.000,E1 14.592} C_DIS
LIN {X -0.022,Y -189.755,Z 1832.058,A 0.000,B 0.000,C 90.000,E1 10.489} C_DIS
LIN {X -0.084,Y -186.798,Z 1832.035,A 0.000,B 0.000,C 90.000,E1 6.372} C_DIS
LIN {X -0.033,Y -184.140,Z 1831.997,A 0.000,B 0.000,C 90.000,E1 359.542} C_DIS
LIN {X 0.049,Y -183.672,Z 1831.960,A 0.000,B 0.000,C 90.000,E1 352.818} C_DIS
LIN {X 0.064,Y -184.877,Z 1831.923,A 0.000,B 0.000,C 90.000,E1 346.117} C_DIS
LIN {X -0.062,Y -186.626,Z 1831.895,A 0.000,B 0.000,C 90.000,E1 341.148} C_DIS
LIN {X -0.110,Y -189.271,Z 1831.867,A 0.000,B 0.000,C 90.000,E1 336.177} C_DIS
LIN {X -0.037,Y -192.115,Z 1831.844,A 0.000,B 0.000,C 90.000,E1 332.025} C_DIS
LIN {X -0.089,Y -196.260,Z 1831.817,A 0.000,B 0.000,C 90.000,E1 327.120} C_DIS
LIN {X -0.069,Y -200.261,Z 1831.795,A 0.000,B 0.000,C 90.000,E1 323.050} C_DIS
LIN {X -0.037,Y -205.147,Z 1831.772,A 0.000,B 0.000,C 90.000,E1 319.013} C_DIS
LIN {X -0.045,Y -208.853,Z 1831.759,A 0.000,B 0.000,C 90.000,E1 316.620} C_DIS
LIN {X 0.004,Y -213.548,Z 1831.746,A 0.000,B 0.000,C 90.000,E1 314.231} C_DIS
LIN {X -0.111,Y -217.443,Z 1831.737,A 0.000,B 0.000,C 90.000,E1 312.690} C_DIS
LIN {X 0.002,Y -222.095,Z 1831.728,A 0.000,B 0.000,C 90.000,E1 311.105} C_DIS
LIN {X 0.010,Y -227.565,Z 1831.720,A 0.000,B 0.000,C 90.000,E1 309.564} C_DIS
LIN {X 0.113,Y -233.853,Z 1831.711,A 0.000,B 0.000,C 90.000,E1 308.016} C_DIS
LIN {X -0.031,Y -244.432,Z 1831.699,A 0.000,B 0.000,C 90.000,E1 305.804} C_DIS
LIN {X -0.132,Y -254.188,Z 1831.689,A 0.000,B 0.000,C 90.000,E1 303.992} C_DIS
LIN {X 0.133,Y -264.781,Z 1831.679,A 0.000,B 0.000,C 90.000,E1 302.133} C_DIS
LIN {X 0.132,Y -283.277,Z 1831.663,A 0.000,B 0.000,C 90.000,E1 299.333} C_DIS
LIN {X -0.065,Y -297.790,Z 1831.652,A 0.000,B 0.000,C 90.000,E1 297.334} C_DIS
LIN {X 0.010,Y -312.479,Z 1831.641,A 0.000,B 0.000,C 90.000,E1 295.335} C_DIS
LIN {X 0.099,Y -327.217,Z 1831.630,A 0.000,B 0.000,C 90.000,E1 293.387} C_DIS
LIN {X -0.078,Y -339.277,Z 1831.621,A 0.000,B 0.000,C 90.000,E1 291.844} C_DIS
LIN {X -0.090,Y -348.459,Z 1831.614,A 0.000,B 0.000,C 90.000,E1 290.610} C_DIS
LIN {X -0.030,Y -354.910,Z 1831.609,A 0.000,B 0.000,C 90.000,E1 289.685} C_DIS
LIN {X -0.022,Y -360.848,Z 1831.604,A 0.000,B 0.000,C 90.000,E1 288.779} C_DIS
LIN {X 0.038,Y -366.198,Z 1831.599,A 0.000,B 0.000,C 90.000,E1 287.873} C_DIS
LIN {X 0.073,Y -369.334,Z 1831.596,A 0.000,B 0.000,C 90.000,E1 287.275} C_DIS
LIN {X 0.130,Y -372.080,Z 1831.593,A 0.000,B 0.000,C 90.000,E1 286.677} C_DIS
LIN {X 0.204,Y -374.416,Z 1831.589,A 0.000,B 0.000,C 90.000,E1 286.079} C_DIS
LIN {X -0.068,Y -376.400,Z 1831.586,A 0.000,B 0.000,C 90.000,E1 285.536} C_DIS
LIN {X -0.072,Y -378.070,Z 1831.583,A 0.000,B 0.000,C 90.000,E1 284.954} C_DIS
LIN {X 0.035,Y -379.321,Z 1831.580,A 0.000,B 0.000,C 90.000,E1 284.356} C_DIS
LIN {X 0.060,Y -380.201,Z 1831.577,A 0.000,B 0.000,C 90.000,E1 283.772} C_DIS
LIN {X 0.182,Y -380.678,Z 1831.573,A 0.000,B 0.000,C 90.000,E1 283.175} C_DIS
LIN {X -0.151,Y -380.707,Z 1831.570,A 0.000,B 0.000,C 90.000,E1 282.647} C_DIS
LIN {X -0.108,Y -380.306,Z 1831.567,A 0.000,B 0.000,C 90.000,E1 282.063} C_DIS
LIN {X -0.063,Y -379.454,Z 1831.564,A 0.000,B 0.000,C 90.000,E1 281.478} C_DIS
LIN {X -0.021,Y -378.116,Z 1831.561,A 0.000,B 0.000,C 90.000,E1 280.894} C_DIS
LIN {X 0.016,Y -376.372,Z 1831.557,A 0.000,B 0.000,C 90.000,E1 280.310} C_DIS
LIN {X -0.012,Y -373.052,Z 1831.552,A 0.000,B 0.000,C 90.000,E1 279.443} C_DIS
LIN {X -0.102,Y -365.584,Z 1831.543,A 0.000,B 0.000,C 90.000,E1 277.701} C_DIS
LIN {X 0.135,Y -361.248,Z 1831.538,A 0.000,B 0.000,C 90.000,E1 276.777} C_DIS
LIN {X -0.030,Y -355.975,Z 1831.533,A 0.000,B 0.000,C 90.000,E1 275.910} C_DIS
LIN {X 0.175,Y -351.795,Z 1831.529,A 0.000,B 0.000,C 90.000,E1 275.277} C_DIS
LIN {X 0.006,Y -346.878,Z 1831.526,A 0.000,B 0.000,C 90.000,E1 274.702} C_DIS
LIN {X -0.142,Y -341.340,Z 1831.523,A 0.000,B 0.000,C 90.000,E1 274.131} C_DIS
LIN {X -0.080,Y -335.438,Z 1831.520,A 0.000,B 0.000,C 90.000,E1 273.555} C_DIS
LIN {X -0.094,Y -329.267,Z 1831.517,A 0.000,B 0.000,C 90.000,E1 273.037} C_DIS
LIN {X 0.113,Y -322.917,Z 1831.514,A 0.000,B 0.000,C 90.000,E1 272.522} C_DIS
LIN {X -0.056,Y -316.296,Z 1831.512,A 0.000,B 0.000,C 90.000,E1 272.121} C_DIS
LIN {X 0.100,Y -309.528,Z 1831.510,A 0.000,B 0.000,C 90.000,E1 271.718} C_DIS
LIN {X -0.091,Y -302.367,Z 1831.508,A 0.000,B 0.000,C 90.000,E1 271.432} C_DIS
LIN {X 0.016,Y -294.767,Z 1831.506,A 0.000,B 0.000,C 90.000,E1 271.146} C_DIS
LIN {X -0.058,Y -283.401,Z 1831.505,A 0.000,B 0.000,C 90.000,E1 270.859} C_DIS
LIN {X -0.066,Y -272.208,Z 1831.503,A 0.000,B 0.000,C 90.000,E1 270.630} C_DIS
LIN {X -0.110,Y -246.660,Z 1831.501,A 0.000,B 0.000,C 90.000,E1 270.172} C_DIS
LIN {X -0.097,Y -235.502,Z 1831.500,A 0.000,B 0.000,C 90.000,E1 270.057} C_DIS
LIN {X 0.072,Y -230.448,Z 1831.500,A 0.000,B 0.000,C 90.000,E1 270.000} C_DIS
LIN {X 0.029,Y -181.562,Z 1831.500,A 0.000,B 0.000,C 90.000,E1 270.000} C_DIS
LIN {X 0.007,Y -180.835,Z 1831.472,A 0.000,B 0.000,C 90.000,E1 264.894} C_DIS
LIN {X 0.087,Y -178.942,Z 1831.443,A 0.000,B 0.000,C 90.000,E1 259.803} C_DIS
LIN {X -0.046,Y -175.992,Z 1831.415,A 0.000,B 0.000,C 90.000,E1 254.755} C_DIS
LIN {X 0.069,Y -175.495,Z 1831.411,A 0.000,B 0.000,C 90.000,E1 253.866} C_DIS
LIN {X -0.037,Y -172.238,Z 1831.387,A 0.000,B 0.000,C 90.000,E1 249.625} C_DIS
LIN {X -0.059,Y -171.715,Z 1831.382,A 0.000,B 0.000,C 90.000,E1 248.773} C_DIS
LIN {X 0.026,Y -167.311,Z 1831.353,A 0.000,B 0.000,C 90.000,E1 243.563} C_DIS
LIN {X 0.032,Y -166.691,Z 1831.348,A 0.000,B 0.000,C 90.000,E1 242.692} C_DIS
LIN {X 0.023,Y -162.672,Z 1831.324,A 0.000,B 0.000,C 90.000,E1 238.329} C_DIS
LIN {X -0.004,Y -161.363,Z 1831.314,A 0.000,B 0.000,C 90.000,E1 236.580} C_DIS
LIN {X 0.030,Y -157.356,Z 1831.290,A 0.000,B 0.000,C 90.000,E1 232.145} C_DIS
LIN {X 0.058,Y -155.345,Z 1831.275,A 0.000,B 0.000,C 90.000,E1 229.461} C_DIS
LIN {X -0.012,Y -151.692,Z 1831.250,A 0.000,B 0.000,C 90.000,E1 225.000} C_DIS
LIN {X 0.036,Y -150.554,Z 1831.240,A 0.000,B 0.000,C 90.000,E1 223.176} C_DIS
LIN {X -0.047,Y -147.281,Z 1831.215,A 0.000,B 0.000,C 90.000,E1 218.669} C_DIS
LIN {X 0.040,Y -145.309,Z 1831.194,A 0.000,B 0.000,C 90.000,E1 214.978} C_DIS
LIN {X 0.032,Y -142.400,Z 1831.164,A 0.000,B 0.000,C 90.000,E1 209.461} C_DIS
LIN {X 0.014,Y -141.381,Z 1831.148,A 0.000,B 0.000,C 90.000,E1 206.693} C_DIS
LIN {X 0.056,Y -139.349,Z 1831.112,A 0.000,B 0.000,C 90.000,E1 200.174} C_DIS
LIN {X -0.002,Y -138.787,Z 1831.097,A 0.000,B 0.000,C 90.000,E1 197.402} C_DIS
LIN {X 0.056,Y -138.344,Z 1831.055,A 0.000,B 0.000,C 90.000,E1 189.905} C_DIS
LIN {X -0.063,Y -139.386,Z 1831.008,A 0.000,B 0.000,C 90.000,E1 181.547} C_DIS
LIN {X -0.010,Y -141.283,Z 1830.972,A 0.000,B 0.000,C 90.000,E1 175.008} C_DIS
LIN {X -0.052,Y -142.646,Z 1830.957,A 0.000,B 0.000,C 90.000,E1 172.243} C_DIS
LIN {X 0.039,Y -144.982,Z 1830.931,A 0.000,B 0.000,C 90.000,E1 167.589} C_DIS
LIN {X 0.030,Y -147.610,Z 1830.911,A 0.000,B 0.000,C 90.000,E1 163.921} C_DIS
LIN {X -0.032,Y -150.232,Z 1830.891,A 0.000,B 0.000,C 90.000,E1 160.296} C_DIS
LIN {X -0.017,Y -153.624,Z 1830.870,A 0.000,B 0.000,C 90.000,E1 156.666} C_DIS
LIN {X -0.029,Y -157.040,Z 1830.850,A 0.000,B 0.000,C 90.000,E1 153.076} C_DIS
LIN {X 0.040,Y -161.165,Z 1830.831,A 0.000,B 0.000,C 90.000,E1 149.488} C_DIS
LIN {X -0.017,Y -163.260,Z 1830.821,A 0.000,B 0.000,C 90.000,E1 147.740} C_DIS
LIN {X 0.082,Y -167.699,Z 1830.801,A 0.000,B 0.000,C 90.000,E1 144.196} C_DIS
LIN {X -0.005,Y -171.520,Z 1830.787,A 0.000,B 0.000,C 90.000,E1 141.618} C_DIS
LIN {X 0.038,Y -176.458,Z 1830.768,A 0.000,B 0.000,C 90.000,E1 138.162} C_DIS
LIN {X -0.091,Y -180.754,Z 1830.753,A 0.000,B 0.000,C 90.000,E1 135.648} C_DIS
LIN {X 0.027,Y -186.159,Z 1830.735,A 0.000,B 0.000,C 90.000,E1 132.243} C_DIS
LIN {X 0.092,Y -190.798,Z 1830.721,A 0.000,B 0.000,C 90.000,E1 129.725} C_DIS
LIN {X 0.011,Y -196.555,Z 1830.703,A 0.000,B 0.000,C 90.000,E1 126.457} C_DIS
LIN {X 0.096,Y -201.325,Z 1830.689,A 0.000,B 0.000,C 90.000,E1 123.992} C_DIS
LIN {X 0.025,Y -207.298,Z 1830.671,A 0.000,B 0.000,C 90.000,E1 120.797} C_DIS
LIN {X 0.024,Y -210.551,Z 1830.662,A 0.000,B 0.000,C 90.000,E1 119.205} C_DIS
LIN {X 0.026,Y -216.357,Z 1830.645,A 0.000,B 0.000,C 90.000,E1 116.052} C_DIS
LIN {X -0.067,Y -219.493,Z 1830.636,A 0.000,B 0.000,C 90.000,E1 114.515} C_DIS
LIN {X -0.048,Y -224.035,Z 1830.622,A 0.000,B 0.000,C 90.000,E1 111.897} C_DIS
LIN {X -0.091,Y -283.091,Z 1830.622,A 0.000,B 0.000,C 90.000,E1 111.897} C_DIS
LIN {X 0.025,Y -285.080,Z 1830.621,A 0.000,B 0.000,C 90.000,E1 111.844} C_DIS
LIN {X -0.076,Y -289.665,Z 1830.620,A 0.000,B 0.000,C 90.000,E1 111.642} C_DIS
LIN {X -0.016,Y -292.171,Z 1830.619,A 0.000,B 0.000,C 90.000,E1 111.408} C_DIS
LIN {X -0.161,Y -295.978,Z 1830.616,A 0.000,B 0.000,C 90.000,E1 110.918} C_DIS
LIN {X 0.109,Y -309.209,Z 1830.603,A 0.000,B 0.000,C 90.000,E1 108.544} C_DIS
LIN {X -0.102,Y -323.777,Z 1830.591,A 0.000,B 0.000,C 90.000,E1 106.315} C_DIS
LIN {X -0.060,Y -337.441,Z 1830.580,A 0.000,B 0.000,C 90.000,E1 104.411} C_DIS
LIN {X 0.086,Y -352.290,Z 1830.570,A 0.000,B 0.000,C 90.000,E1 102.535} C_DIS
LIN {X 0.108,Y -370.668,Z 1830.558,A 0.000,B 0.000,C 90.000,E1 100.489} C_DIS
LIN {X 0.152,Y -389.525,Z 1830.548,A 0.000,B 0.000,C 90.000,E1 98.624} C_DIS
LIN {X 0.067,Y -408.727,Z 1830.539,A 0.000,B 0.000,C 90.000,E1 96.947} C_DIS
LIN {X -0.129,Y -431.094,Z 1830.529,A 0.000,B 0.000,C 90.000,E1 95.220} C_DIS
LIN {X 0.009,Y -439.498,Z 1830.526,A 0.000,B 0.000,C 90.000,E1 94.588} C_DIS
LIN {X -0.078,Y -443.297,Z 1830.523,A 0.000,B 0.000,C 90.000,E1 94.188} C_DIS
LIN {X 0.120,Y -444.946,Z 1830.522,A 0.000,B 0.000,C 90.000,E1 93.898} C_DIS
LIN {X -0.157,Y -446.191,Z 1830.520,A 0.000,B 0.000,C 90.000,E1 93.669} C_DIS
LIN {X -0.208,Y -447.741,Z 1830.517,A 0.000,B 0.000,C 90.000,E1 93.151} C_DIS
LIN {X 0.171,Y -448.277,Z 1830.514,A 0.000,B 0.000,C 90.000,E1 92.579} C_DIS
LIN {X 0.116,Y -447.886,Z 1830.512,A 0.000,B 0.000,C 90.000,E1 92.064} C_DIS
LIN {X 0.078,Y -446.515,Z 1830.509,A 0.000,B 0.000,C 90.000,E1 91.547} C_DIS
LIN {X -0.172,Y -445.395,Z 1830.507,A 0.000,B 0.000,C 90.000,E1 91.318} C_DIS
LIN {X -0.042,Y -440.596,Z 1830.503,A 0.000,B 0.000,C 90.000,E1 90.516} C_DIS
LIN {X -0.198,Y -429.067,Z 1830.493,A 0.000,B 0.000,C 90.000,E1 88.682} C_DIS
LIN {X -0.128,Y -417.310,Z 1830.482,A 0.000,B 0.000,C 90.000,E1 86.788} C_DIS
LIN {X 0.108,Y -405.490,Z 1830.471,A 0.000,B 0.000,C 90.000,E1 84.837} C_DIS
LIN {X 0.166,Y -393.557,Z 1830.461,A 0.000,B 0.000,C 90.000,E1 82.875} C_DIS
LIN {X 0.028,Y -381.610,Z 1830.449,A 0.000,B 0.000,C 90.000,E1 80.905} C_DIS
LIN {X 0.078,Y -368.054,Z 1830.437,A 0.000,B 0.000,C 90.000,E1 78.578} C_DIS
LIN {X -0.119,Y -350.404,Z 1830.418,A 0.000,B 0.000,C 90.000,E1 75.338} C_DIS
LIN {X -0.151,Y -338.269,Z 1830.405,A 0.000,B 0.000,C 90.000,E1 72.906} C_DIS
LIN {X -0.152,Y -327.893,Z 1830.393,A 0.000,B 0.000,C 90.000,E1 70.732} C_DIS
LIN {X -0.042,Y -313.527,Z 1830.375,A 0.000,B 0.000,C 90.000,E1 67.539} C_DIS
LIN {X 0.073,Y -302.517,Z 1830.361,A 0.000,B 0.000,C 90.000,E1 64.921} C_DIS
LIN {X -0.114,Y -290.308,Z 1830.344,A 0.000,B 0.000,C 90.000,E1 61.975} C_DIS
LIN {X -0.005,Y -280.951,Z 1830.331,A 0.000,B 0.000,C 90.000,E1 59.587} C_DIS
LIN {X 0.049,Y -271.541,Z 1830.318,A 0.000,B 0.000,C 90.000,E1 57.168} C_DIS
LIN {X -0.098,Y -263.420,Z 1830.306,A 0.000,B 0.000,C 90.000,E1 55.102} C_DIS
LIN {X 0.147,Y -253.818,Z 1830.292,A 0.000,B 0.000,C 90.000,E1 52.557} C_DIS
LIN {X -0.067,Y -244.232,Z 1830.278,A 0.000,B 0.000,C 90.000,E1 50.070} C_DIS
LIN {X -0.113,Y -242.227,Z 1830.275,A 0.000,B 0.000,C 90.000,E1 49.542} C_DIS
LIN {X -0.004,Y -242.212,Z 1830.275,A 0.000,B 0.000,C 90.000,E1 49.504} C_DIS
LIN {X 0.064,Y -246.728,Z 1830.270,A 0.000,B 0.000,C 90.000,E1 48.566} C_DIS
LIN {X -0.125,Y -248.259,Z 1830.268,A 0.000,B 0.000,C 90.000,E1 48.243} C_DIS
LIN {X 0.036,Y -248.832,Z 1830.266,A 0.000,B 0.000,C 90.000,E1 47.838} C_DIS
LIN {X 0.045,Y -248.938,Z 1830.262,A 0.000,B 0.000,C 90.000,E1 47.106} C_DIS
LIN {X 0.044,Y -248.453,Z 1830.258,A 0.000,B 0.000,C 90.000,E1 46.377} C_DIS
LIN {X 0.044,Y -247.661,Z 1830.254,A 0.000,B 0.000,C 90.000,E1 45.648} C_DIS
LIN {X 0.036,Y -245.568,Z 1830.246,A 0.000,B 0.000,C 90.000,E1 44.190} C_DIS
LIN {X 0.000,Y -243.030,Z 1830.237,A 0.000,B 0.000,C 90.000,E1 42.732} C_DIS
LIN {X -0.083,Y -238.782,Z 1830.225,A 0.000,B 0.000,C 90.000,E1 40.539} C_DIS
LIN {X -0.060,Y -234.286,Z 1830.213,A 0.000,B 0.000,C 90.000,E1 38.302} C_DIS
LIN {X 0.097,Y -229.569,Z 1830.200,A 0.000,B 0.000,C 90.000,E1 36.011} C_DIS
LIN {X -0.038,Y -223.304,Z 1830.183,A 0.000,B 0.000,C 90.000,E1 33.007} C_DIS
LIN {X 0.092,Y -218.560,Z 1830.171,A 0.000,B 0.000,C 90.000,E1 30.669} C_DIS
LIN {X 0.021,Y -211.014,Z 1830.149,A 0.000,B 0.000,C 90.000,E1 26.796} C_DIS
LIN {X 0.002,Y -205.449,Z 1830.131,A 0.000,B 0.000,C 90.000,E1 23.643} C_DIS
LIN {X 0.065,Y -200.593,Z 1830.114,A 0.000,B 0.000,C 90.000,E1 20.429} C_DIS
LIN {X 0.064,Y -195.264,Z 1830.091,A 0.000,B 0.000,C 90.000,E1 16.386} C_DIS
LIN {X 0.060,Y -190.962,Z 1830.068,A 0.000,B 0.000,C 90.000,E1 12.299} C_DIS
LIN {X 0.092,Y -187.557,Z 1830.046,A 0.000,B 0.000,C 90.000,E1 8.163} C_DIS
LIN {X 0.052,Y -184.520,Z 1830.013,A 0.000,B 0.000,C 90.000,E1 2.350} C_DIS
LIN {X -0.040,Y -183.258,Z 1829.974,A 0.000,B 0.000,C 90.000,E1 355.355} C_DIS
LIN {X -0.046,Y -184.096,Z 1829.932,A 0.000,B 0.000,C 90.000,E1 347.813} C_DIS
LIN {X 0.008,Y -185.624,Z 1829.904,A 0.000,B 0.000,C 90.000,E1 342.779} C_DIS
LIN {X -0.067,Y -188.475,Z 1829.872,A 0.000,B 0.000,C 90.000,E1 336.975} C_DIS
LIN {X 0.057,Y -191.832,Z 1829.844,A 0.000,B 0.000,C 90.000,E1 331.975} C_DIS
LIN {X 0.096,Y -196.012,Z 1829.817,A 0.000,B 0.000,C 90.000,E1 327.041} C_DIS
LIN {X -0.005,Y -200.043,Z 1829.794,A 0.000,B 0.000,C 90.000,E1 323.004} C_DIS
LIN {X -0.007,Y -205.039,Z 1829.772,A 0.000,B 0.000,C 90.000,E1 318.976} C_DIS
LIN {X -0.010,Y -208.816,Z 1829.759,A 0.000,B 0.000,C 90.000,E1 316.581} C_DIS
LIN {X 0.046,Y -213.597,Z 1829.746,A 0.000,B 0.000,C 90.000,E1 314.190} C_DIS
LIN {X 0.085,Y -217.556,Z 1829.737,A 0.000,B 0.000,C 90.000,E1 312.609} C_DIS
LIN {X 0.035,Y -222.263,Z 1829.728,A 0.000,B 0.000,C 90.000,E1 311.067} C_DIS
LIN {X -0.105,Y -227.784,Z 1829.720,A 0.000,B 0.000,C 90.000,E1 309.564} C_DIS
LIN {X -0.002,Y -234.109,Z 1829.711,A 0.000,B 0.000,C 90.000,E1 308.016} C_DIS
LIN {X -0.146,Y -244.730,Z 1829.699,A 0.000,B 0.000,C 90.000,E1 305.804} C_DIS
LIN {X -0.025,Y -256.582,Z 1829.687,A 0.000,B 0.000,C 90.000,E1 303.579} C_DIS
LIN {X 0.057,Y -269.652,Z 1829.675,A 0.000,B 0.000,C 90.000,E1 301.416} C_DIS
LIN {X -0.021,Y -286.097,Z 1829.661,A 0.000,B 0.000,C 90.000,E1 298.999} C_DIS
LIN {X 0.094,Y -300.681,Z 1829.650,A 0.000,B 0.000,C 90.000,E1 296.950} C_DIS
LIN {X -0.093,Y -313.001,Z 1829.641,A 0.000,B 0.000,C 90.000,E1 295.335} C_DIS
LIN {X 0.062,Y -325.344,Z 1829.632,A 0.000,B 0.000,C 90.000,E1 293.695} C_DIS
LIN {X -0.153,Y -337.496,Z 1829.623,A 0.000,B 0.000,C 90.000,E1 292.153} C_DIS
LIN {X -0.189,Y -346.876,Z 1829.616,A 0.000,B 0.000,C 90.000,E1 290.918} C_DIS
LIN {X -0.137,Y -353.483,Z 1829.611,A 0.000,B 0.000,C 90.000,E1 289.993} C_DIS
LIN {X -0.151,Y -359.583,Z 1829.606,A 0.000,B 0.000,C 90.000,E1 289.087} C_DIS
LIN {X -0.096,Y -365.156,Z 1829.601,A 0.000,B 0.000,C 90.000,E1 288.181} C_DIS
LIN {X -0.070,Y -368.476,Z 1829.598,A 0.000,B 0.000,C 90.000,E1 287.583} C_DIS
LIN {X 0.066,Y -372.701,Z 1829.593,A 0.000,B 0.000,C 90.000,E1 286.677} C_DIS
LIN {X 0.144,Y -375.032,Z 1829.589,A 0.000,B 0.000,C 90.000,E1 286.079} C_DIS
LIN {X -0.126,Y -376.992,Z 1829.586,A 0.000,B 0.000,C 90.000,E1 285.536} C_DIS
LIN {X -0.126,Y -378.634,Z 1829.583,A 0.000,B 0.000,C 90.000,E1 284.954} C_DIS
LIN {X -0.015,Y -379.873,Z 1829.580,A 0.000,B 0.000,C 90.000,E1 284.356} C_DIS
LIN {X 0.012,Y -380.734,Z 1829.577,A 0.000,B 0.000,C 90.000,E1 283.772} C_DIS
LIN {X 0.138,Y -381.203,Z 1829.573,A 0.000,B 0.000,C 90.000,E1 283.175} C_DIS
LIN {X 0.180,Y -381.167,Z 1829.570,A 0.000,B 0.000,C 90.000,E1 282.591} C_DIS
LIN {X -0.145,Y -380.788,Z 1829.567,A 0.000,B 0.000,C 90.000,E1 282.063} C_DIS
LIN {X -0.098,Y -379.903,Z 1829.564,A 0.000,B 0.000,C 90.000,E1 281.478} C_DIS
LIN {X -0.052,Y -378.582,Z 1829.560,A 0.000,B 0.000,C 90.000,E1 280.894} C_DIS
LIN {X -0.014,Y -376.813,Z 1829.557,A 0.000,B 0.000,C 90.000,E1 280.310} C_DIS
LIN {X -0.037,Y -373.505,Z 1829.552,A 0.000,B 0.000,C 90.000,E1 279.443} C_DIS
LIN {X -0.101,Y -367.267,Z 1829.544,A 0.000,B 0.000,C 90.000,E1 277.992} C_DIS
LIN {X 0.151,Y -363.066,Z 1829.539,A 0.000,B 0.000,C 90.000,E1 277.068} C_DIS
LIN {X 0.086,Y -359.867,Z 1829.536,A 0.000,B 0.000,C 90.000,E1 276.486} C_DIS
LIN {X -0.040,Y -356.205,Z 1829.533,A 0.000,B 0.000,C 90.000,E1 275.910} C_DIS
LIN {X 0.168,Y -351.966,Z 1829.529,A 0.000,B 0.000,C 90.000,E1 275.277} C_DIS
LIN {X 0.000,Y -347.077,Z 1829.526,A 0.000,B 0.000,C 90.000,E1 274.702} C_DIS
LIN {X -0.150,Y -341.511,Z 1829.523,A 0.000,B 0.000,C 90.000,E1 274.131} C_DIS
LIN {X -0.092,Y -335.594,Z 1829.520,A 0.000,B 0.000,C 90.000,E1 273.555} C_DIS
LIN {X -0.118,Y -329.423,Z 1829.517,A 0.000,B 0.000,C 90.000,E1 273.037} C_DIS
LIN {X 0.113,Y -323.044,Z 1829.514,A 0.000,B 0.000,C 90.000,E1 272.522} C_DIS
LIN {X -0.031,Y -316.489,Z 1829.512,A 0.000,B 0.000,C 90.000,E1 272.121} C_DIS
LIN {X 0.112,Y -309.595,Z 1829.510,A 0.000,B 0.000,C 90.000,E1 271.718} C_DIS
LIN {X -0.088,Y -302.431,Z 1829.508,A 0.000,B 0.000,C 90.000,E1 271.432} C_DIS
LIN {X 0.015,Y -294.673,Z 1829.506,A 0.000,B 0.000,C 90.000,E1 271.146} C_DIS
LIN {X -0.086,Y -283.124,Z 1829.505,A 0.000,B 0.000,C 90.000,E1 270.859} C_DIS
LIN {X -0.092,Y -271.836,Z 1829.503,A 0.000,B 0.000,C 90.000,E1 270.630} C_DIS
LIN {X -0.103,Y -250.074,Z 1829.501,A 0.000,B 0.000,C 90.000,E1 270.229} C_DIS
LIN {X 0.091,Y -240.595,Z 1829.500,A 0.000,B 0.000,C 90.000,E1 270.057} C_DIS
LIN {X 0.113,Y -229.623,Z 1829.500,A 0.000,B 0.000,C 90.000,E1 270.000} C_DIS
LIN {X 0.062,Y -181.564,Z 1829.500,A 0.000,B 0.000,C 90.000,E1 270.000} C_DIS
LIN {X -0.009,Y -180.907,Z 1829.475,A 0.000,B 0.000,C 90.000,E1 265.469} C_DIS
LIN {X 0.048,Y -180.735,Z 1829.470,A 0.000,B 0.000,C 90.000,E1 264.609} C_DIS
LIN {X -0.031,Y -178.825,Z 1829.442,A 0.000,B 0.000,C 90.000,E1 259.567} C_DIS
LIN {X 0.051,Y -175.869,Z 1829.414,A 0.000,B 0.000,C 90.000,E1 254.448} C_DIS
LIN {X 0.045,Y -173.840,Z 1829.400,A 0.000,B 0.000,C 90.000,E1 251.891} C_DIS
LIN {X 0.034,Y -171.508,Z 1829.380,A 0.000,B 0.000,C 90.000,E1 248.465} C_DIS
LIN {X 0.020,Y -167.736,Z 1829.356,A 0.000,B 0.000,C 90.000,E1 244.152} C_DIS
LIN {X 0.036,Y -166.434,Z 1829.347,A 0.000,B 0.000,C 90.000,E1 242.410} C_DIS
LIN {X -0.050,Y -163.153,Z 1829.327,A 0.000,B 0.000,C 90.000,E1 238.948} C_DIS
LIN {X -0.001,Y -161.109,Z 1829.313,A 0.000,B 0.000,C 90.000,E1 236.294} C_DIS
LIN {X -0.017,Y -157.835,Z 1829.293,A 0.000,B 0.000,C 90.000,E1 232.763} C_DIS
LIN {X 0.046,Y -155.868,Z 1829.278,A 0.000,B 0.000,C 90.000,E1 230.070} C_DIS
LIN {X -0.005,Y -152.118,Z 1829.253,A 0.000,B 0.000,C 90.000,E1 225.607} C_DIS
LIN {X 0.009,Y -150.368,Z 1829.238,A 0.000,B 0.000,C 90.000,E1 222.894} C_DIS
LIN {X -0.069,Y -147.102,Z 1829.213,A 0.000,B 0.000,C 90.000,E1 218.382} C_DIS
LIN {X 0.041,Y -145.671,Z 1829.198,A 0.000,B 0.000,C 90.000,E1 215.598} C_DIS
LIN {X 0.044,Y -143.053,Z 1829.172,A 0.000,B 0.000,C 90.000,E1 211.003} C_DIS
LIN {X -0.021,Y -141.675,Z 1829.152,A 0.000,B 0.000,C 90.000,E1 207.334} C_DIS
LIN {X -0.042,Y -139.454,Z 1829.116,A 0.000,B 0.000,C 90.000,E1 200.844} C_DIS
LIN {X 0.009,Y -139.189,Z 1829.105,A 0.000,B 0.000,C 90.000,E1 198.960} C_DIS
LIN {X 0.033,Y -138.323,Z 1829.053,A 0.000,B 0.000,C 90.000,E1 189.613} C_DIS
LIN {X 0.040,Y -139.458,Z 1829.007,A 0.000,B 0.000,C 90.000,E1 181.203} C_DIS
LIN {X -0.020,Y -141.010,Z 1828.976,A 0.000,B 0.000,C 90.000,E1 175.641} C_DIS
LIN {X 0.071,Y -142.764,Z 1828.955,A 0.000,B 0.000,C 90.000,E1 171.894} C_DIS
LIN {X 0.026,Y -145.172,Z 1828.929,A 0.000,B 0.000,C 90.000,E1 167.297} C_DIS
LIN {X 0.060,Y -147.794,Z 1828.909,A 0.000,B 0.000,C 90.000,E1 163.614} C_DIS
LIN {X -0.045,Y -150.477,Z 1828.889,A 0.000,B 0.000,C 90.000,E1 160.007} C_DIS
LIN {X 0.029,Y -153.930,Z 1828.869,A 0.000,B 0.000,C 90.000,E1 156.357} C_DIS
LIN {X -0.048,Y -157.342,Z 1828.849,A 0.000,B 0.000,C 90.000,E1 152.794} C_DIS
LIN {X 0.036,Y -161.535,Z 1828.829,A 0.000,B 0.000,C 90.000,E1 149.203} C_DIS
LIN {X 0.049,Y -165.734,Z 1828.809,A 0.000,B 0.000,C 90.000,E1 145.674} C_DIS
LIN {X 0.036,Y -170.685,Z 1828.790,A 0.000,B 0.000,C 90.000,E1 142.190} C_DIS
LIN {X -0.052,Y -175.559,Z 1828.771,A 0.000,B 0.000,C 90.000,E1 138.771} C_DIS
LIN {X 0.068,Y -181.177,Z 1828.752,A 0.000,B 0.000,C 90.000,E1 135.324} C_DIS
LIN {X -0.063,Y -186.635,Z 1828.733,A 0.000,B 0.000,C 90.000,E1 132.000} C_DIS
LIN {X 0.007,Y -191.242,Z 1828.719,A 0.000,B 0.000,C 90.000,E1 129.483} C_DIS
LIN {X -0.071,Y -197.060,Z 1828.701,A 0.000,B 0.000,C 90.000,E1 126.217} C_DIS
LIN {X 0.011,Y -200.333,Z 1828.692,A 0.000,B 0.000,C 90.000,E1 124.565} C_DIS
LIN {X 0.017,Y -207.823,Z 1828.670,A 0.000,B 0.000,C 90.000,E1 120.541} C_DIS
LIN {X 0.023,Y -210.987,Z 1828.661,A 0.000,B 0.000,C 90.000,E1 118.949} C_DIS
LIN {X 0.038,Y -216.867,Z 1828.643,A 0.000,B 0.000,C 90.000,E1 115.796} C_DIS
LIN {X -0.009,Y -218.485,Z 1828.639,A 0.000,B 0.000,C 90.000,E1 115.027} C_DIS
LIN {X 0.009,Y -222.551,Z 1828.626,A 0.000,B 0.000,C 90.000,E1 112.695} C_DIS
LIN {X -0.056,Y -224.038,Z 1828.622,A 0.000,B 0.000,C 90.000,E1 111.897} C_DIS
LIN {X -0.107,Y -283.695,Z 1828.622,A 0.000,B 0.000,C 90.000,E1 111.897} C_DIS
LIN {X -0.019,Y -285.470,Z 1828.621,A 0.000,B 0.000,C 90.000,E1 111.844} C_DIS
LIN {X 0.082,Y -291.230,Z 1828.619,A 0.000,B 0.000,C 90.000,E1 111.482} C_DIS
LIN {X 0.018,Y -294.233,Z 1828.618,A 0.000,B 0.000,C 90.000,E1 111.153} C_DIS
LIN {X -0.015,Y -296.237,Z 1828.616,A 0.000,B 0.000,C 90.000,E1 110.844} C_DIS
LIN {X -0.016,Y -309.348,Z 1828.603,A 0.000,B 0.000,C 90.000,E1 108.544} C_DIS
LIN {X 0.089,Y -323.921,Z 1828.590,A 0.000,B 0.000,C 90.000,E1 106.260} C_DIS
LIN {X 0.144,Y -337.598,Z 1828.580,A 0.000,B 0.000,C 90.000,E1 104.356} C_DIS
LIN {X -0.039,Y -352.460,Z 1828.570,A 0.000,B 0.000,C 90.000,E1 102.535} C_DIS
LIN {X -0.025,Y -370.864,Z 1828.558,A 0.000,B 0.000,C 90.000,E1 100.489} C_DIS
LIN {X 0.047,Y -389.688,Z 1828.548,A 0.000,B 0.000,C 90.000,E1 98.624} C_DIS
LIN {X -0.055,Y -408.929,Z 1828.539,A 0.000,B 0.000,C 90.000,E1 96.947} C_DIS
LIN {X 0.185,Y -431.298,Z 1828.529,A 0.000,B 0.000,C 90.000,E1 95.163} C_DIS
LIN {X -0.083,Y -439.638,Z 1828.525,A 0.000,B 0.000,C 90.000,E1 94.588} C_DIS
LIN {X 0.133,Y -441.696,Z 1828.524,A 0.000,B 0.000,C 90.000,E1 94.359} C_DIS
LIN {X -0.027,Y -443.641,Z 1828.523,A 0.000,B 0.000,C 90.000,E1 94.131} C_DIS
LIN {X -0.156,Y -445.126,Z 1828.521,A 0.000,B 0.000,C 90.000,E1 93.898} C_DIS
LIN {X 0.023,Y -446.316,Z 1828.520,A 0.000,B 0.000,C 90.000,E1 93.612} C_DIS
LIN {X 0.205,Y -447.191,Z 1828.519,A 0.000,B 0.000,C 90.000,E1 93.326} C_DIS
LIN {X 0.162,Y -448.146,Z 1828.516,A 0.000,B 0.000,C 90.000,E1 92.808} C_DIS
LIN {X 0.102,Y -448.156,Z 1828.513,A 0.000,B 0.000,C 90.000,E1 92.293} C_DIS
LIN {X 0.065,Y -447.227,Z 1828.510,A 0.000,B 0.000,C 90.000,E1 91.776} C_DIS
LIN {X 0.012,Y -445.209,Z 1828.507,A 0.000,B 0.000,C 90.000,E1 91.260} C_DIS
LIN {X 0.052,Y -437.057,Z 1828.500,A 0.000,B 0.000,C 90.000,E1 89.943} C_DIS
LIN {X 0.115,Y -427.177,Z 1828.491,A 0.000,B 0.000,C 90.000,E1 88.339} C_DIS
LIN {X 0.136,Y -415.402,Z 1828.480,A 0.000,B 0.000,C 90.000,E1 86.445} C_DIS
LIN {X -0.046,Y -403.546,Z 1828.470,A 0.000,B 0.000,C 90.000,E1 84.546} C_DIS
LIN {X -0.068,Y -391.614,Z 1828.459,A 0.000,B 0.000,C 90.000,E1 82.591} C_DIS
LIN {X 0.127,Y -379.656,Z 1828.448,A 0.000,B 0.000,C 90.000,E1 80.566} C_DIS
LIN {X 0.173,Y -364.515,Z 1828.433,A 0.000,B 0.000,C 90.000,E1 77.937} C_DIS
LIN {X -0.064,Y -347.111,Z 1828.415,A 0.000,B 0.000,C 90.000,E1 74.685} C_DIS
LIN {X -0.078,Y -335.072,Z 1828.401,A 0.000,B 0.000,C 90.000,E1 72.236} C_DIS
LIN {X 0.122,Y -323.289,Z 1828.387,A 0.000,B 0.000,C 90.000,E1 69.699} C_DIS
LIN {X -0.090,Y -309.171,Z 1828.370,A 0.000,B 0.000,C 90.000,E1 66.538} C_DIS
